LIN {X 0,Y 226.973,Z 1141.25,A -85,B 0,C 180,E1 10854.134,E2 10854.134} C_VEL
LIN {X 0,Y 235.059,Z 1134.942,A -85,B 0,C 180,E1 10847.384,E2 10847.384} C_VEL
LIN {X 0,Y 243.394,Z 1128.553,A -85,B 0,C 180,E1 10842.316,E2 10842.316} C_VEL
LIN {X 0,Y 253.409,Z 1120.828,A -85,B 0,C 180,E1 10837.527,E2 10837.527} C_VEL
LIN {X 0,Y 267.885,Z 1109.245,A -85,B 0,C 180,E1 10832.085,E2 10832.085} C_VEL
LIN {X 0,Y 280.211,Z 1098.882,A -85,B 0,C 180,E1 10828.333,E2 10828.333} C_VEL
LIN {X 0,Y 293.347,Z 1087.293,A -85,B 0,C 180,E1 10824.954,E2 10824.954} C_VEL
LIN {X 0,Y 310.134,Z 1071.349,A -85,B 0,C 180,E1 10821.295,E2 10821.295} C_VEL
LIN {X 0,Y 323.853,Z 1057.227,A -85,B 0,C 180,E1 10818.729,E2 10818.729} C_VEL
LIN {X 0,Y 337.044,Z 1042.652,A -85,B 0,C 180,E1 10816.547,E2 10816.547} C_VEL
LIN {X 0,Y 352.779,Z 1023.717,A -85,B 0,C 180,E1 10814.232,E2 10814.232} C_VEL
LIN {X 0,Y 366.214,Z 1005.755,A -85,B 0,C 180,E1 10812.456,E2 10812.456} C_VEL
LIN {X 0,Y 377.493,Z 989.298,A -85,B 0,C 180,E1 10811.087,E2 10811.087} C_VEL
LIN {X 0,Y 389.316,Z 970.374,A -85,B 0,C 180,E1 10809.759,E2 10809.759} C_VEL
LIN {X 0,Y 402.725,Z 946.04,A -85,B 0,C 180,E1 10808.363,E2 10808.363} C_VEL
LIN {X 0,Y 411.936,Z 927.031,A -85,B 0,C 180,E1 10807.468,E2 10807.468} C_VEL
LIN {X 0,Y 420.462,Z 907.175,A -85,B 0,C 180,E1 10806.669,E2 10806.669} C_VEL
LIN {X 0,Y 429.627,Z 882.607,A -85,B 0,C 180,E1 10805.851,E2 10805.851} C_VEL
LIN {X 0,Y 437.317,Z 856.996,A -85,B 0,C 180,E1 10805.178,E2 10805.178} C_VEL
LIN {X 0,Y 442.393,Z 836.475,A -85,B 0,C 180,E1 10804.748,E2 10804.748} C_VEL
LIN {X 0,Y 446.869,Z 813.721,A -85,B 0,C 180,E1 10804.357,E2 10804.357} C_VEL
LIN {X 0,Y 451.545,Z 778.74,A -85,B 0,C 180,E1 10803.872,E2 10803.872} C_VEL
LIN {X 0,Y 453.629,Z 760.255,A -85,B 0,C 180,E1 10803.626,E2 10803.626} C_VEL
LIN {X 0,Y 454.379,Z 752.732,A -85,B 0,C 180,E1 10803.403,E2 10803.403} C_VEL
LIN {X 0,Y 456.025,Z 733.241,A -85,B 0,C 180,E1 10802.357,E2 10802.357} C_VEL
LIN {X 0,Y 456.71,Z 726.771,A -85,B 0,C 180,E1 10802.178,E2 10802.178} C_VEL
LIN {X 0,Y 468.964,Z 621.482,A -85,B 0,C 180,E1 10800.794,E2 10800.794} C_VEL
LIN {X 0,Y 468.493,Z 619.747,A -85,B 0,C 180,E1 10797.798,E2 10797.798} C_VEL
LIN {X 0,Y 469.144,Z 622.007,A -85,B 0,C 180,E1 10794.232,E2 10794.232} C_VEL
LIN {X 0,Y 447.711,Z 806.552,A -85,B 0,C 180,E1 10791.736,E2 10791.736} C_VEL
LIN {X 0,Y 443.092,Z 833.793,A -85,B 0,C 180,E1 10791.332,E2 10791.332} C_VEL
LIN {X 0,Y 436.841,Z 859.788,A -85,B 0,C 180,E1 10790.9,E2 10790.9} C_VEL
LIN {X 0,Y 430.614,Z 880.919,A -85,B 0,C 180,E1 10790.485,E2 10790.485} C_VEL
LIN {X 0,Y 422.897,Z 903.181,A -85,B 0,C 180,E1 10789.937,E2 10789.937} C_VEL
LIN {X 0,Y 411.827,Z 930.087,A -85,B 0,C 180,E1 10789.097,E2 10789.097} C_VEL
LIN {X 0,Y 401.901,Z 950.938,A -85,B 0,C 180,E1 10788.281,E2 10788.281} C_VEL
LIN {X 0,Y 391.891,Z 969.818,A -85,B 0,C 180,E1 10787.395,E2 10787.395} C_VEL
LIN {X 0,Y 379.849,Z 990.376,A -85,B 0,C 180,E1 10786.24,E2 10786.24} C_VEL
LIN {X 0,Y 364.513,Z 1013.698,A -85,B 0,C 180,E1 10784.615,E2 10784.615} C_VEL
LIN {X 0,Y 351.656,Z 1031.443,A -85,B 0,C 180,E1 10783.091,E2 10783.091} C_VEL
LIN {X 0,Y 339.49,Z 1047.003,A -85,B 0,C 180,E1 10781.504,E2 10781.504} C_VEL
LIN {X 0,Y 325.202,Z 1064.029,A -85,B 0,C 180,E1 10779.424,E2 10779.424} C_VEL
LIN {X 0,Y 307.386,Z 1083.642,A -85,B 0,C 180,E1 10776.415,E2 10776.415} C_VEL
LIN {X 0,Y 293.416,Z 1097.967,A -85,B 0,C 180,E1 10773.665,E2 10773.665} C_VEL
LIN {X 0,Y 280.033,Z 1111.045,A -85,B 0,C 180,E1 10770.599,E2 10770.599} C_VEL
LIN {X 0,Y 265.034,Z 1125.203,A -85,B 0,C 180,E1 10766.485,E2 10766.485} C_VEL
LIN {X 0,Y 250.118,Z 1138.668,A -85,B 0,C 180,E1 10761.418,E2 10761.418} C_VEL
LIN {X 0,Y 239.086,Z 1148.595,A -85,B 0,C 180,E1 10756.691,E2 10756.691} C_VEL
LIN {X 0,Y 229.528,Z 1157.411,A -85,B 0,C 180,E1 10751.463,E2 10751.463} C_VEL
LIN {X 0,Y 219.97,Z 1166.782,A -85,B 0,C 180,E1 10744.308,E2 10744.308} C_VEL
LIN {X 0,Y 214.19,Z 1173.147,A -85,B 0,C 180,E1 10737.828,E2 10737.828} C_VEL
LIN {X 0,Y 210.917,Z 1177.583,A -85,B 0,C 180,E1 10731.994,E2 10731.994} C_VEL
LIN {X 0,Y 209.151,Z 1180.939,A -85,B 0,C 180,E1 10726.098,E2 10726.098} C_VEL
LIN {X 0,Y 208.563,Z 1183.075,A -85,B 0,C 180,E1 10720.638,E2 10720.638} C_VEL
LIN {X 0,Y 208.6,Z 1184.174,A -85,B 0,C 180,E1 10715.777,E2 10715.777} C_VEL
LIN {X 0,Y 208.736,Z 1184.477,A -85,B 0,C 180,E1 10711.098,E2 10711.098} C_VEL
LIN {X 0,Y 208.696,Z 1183.922,A -85,B 0,C 180,E1 10706.154,E2 10706.154} C_VEL
LIN {X 0,Y 208.612,Z 1182.339,A -85,B 0,C 180,E1 10700.886,E2 10700.886} C_VEL
LIN {X 0,Y 209.086,Z 1179.246,A -85,B 0,C 180,E1 10694.751,E2 10694.751} C_VEL
LIN {X 0,Y 210.519,Z 1175.309,A -85,B 0,C 180,E1 10689.132,E2 10689.132} C_VEL
LIN {X 0,Y 213.256,Z 1170.278,A -85,B 0,C 180,E1 10683.551,E2 10683.551} C_VEL
LIN {X 0,Y 217.415,Z 1164.128,A -85,B 0,C 180,E1 10678.071,E2 10678.071} C_VEL
LIN {X 0,Y 223.422,Z 1156.436,A -85,B 0,C 180,E1 10672.51,E2 10672.51} C_VEL
LIN {X 0,Y 233.164,Z 1145.065,A -85,B 0,C 180,E1 10665.998,E2 10665.998} C_VEL
LIN {X 0,Y 243.301,Z 1133.621,A -85,B 0,C 180,E1 10660.874,E2 10660.874} C_VEL
LIN {X 0,Y 253.371,Z 1122.401,A -85,B 0,C 180,E1 10656.767,E2 10656.767} C_VEL
LIN {X 0,Y 266.019,Z 1108.199,A -85,B 0,C 180,E1 10652.514,E2 10652.514} C_VEL
LIN {X 0,Y 280.155,Z 1091.564,A -85,B 0,C 180,E1 10648.572,E2 10648.572} C_VEL
LIN {X 0,Y 291.973,Z 1077.025,A -85,B 0,C 180,E1 10645.758,E2 10645.758} C_VEL
LIN {X 0,Y 303.945,Z 1061.531,A -85,B 0,C 180,E1 10643.251,E2 10643.251} C_VEL
LIN {X 0,Y 318.505,Z 1041.486,A -85,B 0,C 180,E1 10640.586,E2 10640.586} C_VEL
LIN {X 0,Y 331.631,Z 1021.599,A -85,B 0,C 180,E1 10638.456,E2 10638.456} C_VEL
LIN {X 0,Y 342.65,Z 1003.559,A -85,B 0,C 180,E1 10636.842,E2 10636.842} C_VEL
LIN {X 0,Y 354.044,Z 983.305,A -85,B 0,C 180,E1 10635.328,E2 10635.328} C_VEL
LIN {X 0,Y 366.538,Z 958.361,A -85,B 0,C 180,E1 10633.806,E2 10633.806} C_VEL
LIN {X 0,Y 375.614,Z 937.919,A -85,B 0,C 180,E1 10632.788,E2 10632.788} C_VEL
LIN {X 0,Y 383.742,Z 917.39,A -85,B 0,C 180,E1 10631.936,E2 10631.936} C_VEL
LIN {X 0,Y 392.509,Z 892.087,A -85,B 0,C 180,E1 10631.078,E2 10631.078} C_VEL
LIN {X 0,Y 399.826,Z 866.079,A -85,B 0,C 180,E1 10630.401,E2 10630.401} C_VEL
LIN {X 0,Y 404.934,Z 844.022,A -85,B 0,C 180,E1 10629.944,E2 10629.944} C_VEL
LIN {X 0,Y 409.416,Z 818.913,A -85,B 0,C 180,E1 10629.487,E2 10629.487} C_VEL
LIN {X 0,Y 413.661,Z 781.521,A -85,B 0,C 180,E1 10628.913,E2 10628.913} C_VEL
LIN {X 0,Y 432.506,Z 593.201,A -85,B 0,C 180,E1 10626.162,E2 10626.162} C_VEL
LIN {X 0,Y 429.414,Z 586.105,A -85,B 0,C 180,E1 10623.605,E2 10623.605} C_VEL
LIN {X 0,Y 427.117,Z 580.871,A -85,B 0,C 180,E1 10621.207,E2 10621.207} C_VEL
LIN {X 0,Y 425.896,Z 578.251,A -85,B 0,C 180,E1 10619.596,E2 10619.596} C_VEL
LIN {X 0,Y 424.641,Z 575.258,A -85,B 0,C 180,E1 10617.301,E2 10617.301} C_VEL
LIN {X 0,Y 423.647,Z 573.176,A -85,B 0,C 180,E1 10613.223,E2 10613.223} C_VEL
LIN {X 0,Y 423.893,Z 573.926,A -85,B 0,C 180,E1 10610.496,E2 10610.496} C_VEL
LIN {X 0,Y 424.964,Z 575.871,A -85,B 0,C 180,E1 10607.705,E2 10607.705} C_VEL
LIN {X 0,Y 426.778,Z 579.948,A -85,B 0,C 180,E1 10604.926,E2 10604.926} C_VEL
LIN {X 0,Y 429.137,Z 585.108,A -85,B 0,C 180,E1 10602.368,E2 10602.368} C_VEL
LIN {X 0,Y 430.931,Z 589.439,A -85,B 0,C 180,E1 10600.767,E2 10600.767} C_VEL
LIN {X 0,Y 409.317,Z 799.134,A -85,B 0,C 180,E1 10597.801,E2 10597.801} C_VEL
LIN {X 0,Y 405.219,Z 825.67,A -85,B 0,C 180,E1 10597.343,E2 10597.343} C_VEL
LIN {X 0,Y 399.741,Z 850.636,A -85,B 0,C 180,E1 10596.777,E2 10596.777} C_VEL
LIN {X 0,Y 394.029,Z 871.901,A -85,B 0,C 180,E1 10596.174,E2 10596.174} C_VEL
LIN {X 0,Y 386.657,Z 895.114,A -85,B 0,C 180,E1 10595.36,E2 10595.36} C_VEL
LIN {X 0,Y 377.297,Z 919.717,A -85,B 0,C 180,E1 10594.292,E2 10594.292} C_VEL
LIN {X 0,Y 368.832,Z 939.096,A -85,B 0,C 180,E1 10593.282,E2 10593.282} C_VEL
LIN {X 0,Y 359.283,Z 958.656,A -85,B 0,C 180,E1 10592.077,E2 10592.077} C_VEL
LIN {X 0,Y 346.794,Z 981.508,A -85,B 0,C 180,E1 10590.373,E2 10590.373} C_VEL
LIN {X 0,Y 334.96,Z 1000.727,A -85,B 0,C 180,E1 10588.617,E2 10588.617} C_VEL
LIN {X 0,Y 323.806,Z 1017.378,A -85,B 0,C 180,E1 10586.804,E2 10586.804} C_VEL
LIN {X 0,Y 310.836,Z 1035.283,A -85,B 0,C 180,E1 10584.47,E2 10584.47} C_VEL
LIN {X 0,Y 296.991,Z 1052.66,A -85,B 0,C 180,E1 10581.667,E2 10581.667} C_VEL
LIN {X 0,Y 285.132,Z 1066.573,A -85,B 0,C 180,E1 10578.932,E2 10578.932} C_VEL
LIN {X 0,Y 273.308,Z 1079.709,A -85,B 0,C 180,E1 10575.81,E2 10575.81} C_VEL
LIN {X 0,Y 258.957,Z 1094.789,A -85,B 0,C 180,E1 10571.319,E2 10571.319} C_VEL
LIN {X 0,Y 248.09,Z 1105.699,A -85,B 0,C 180,E1 10567.195,E2 10567.195} C_VEL
LIN {X 0,Y 238.437,Z 1115.241,A -85,B 0,C 180,E1 10562.748,E2 10562.748} C_VEL
LIN {X 0,Y 228.33,Z 1125.281,A -85,B 0,C 180,E1 10556.81,E2 10556.81} C_VEL
LIN {X 0,Y 220.905,Z 1132.814,A -85,B 0,C 180,E1 10550.951,E2 10550.951} C_VEL
LIN {X 0,Y 215.987,Z 1138.253,A -85,B 0,C 180,E1 10545.575,E2 10545.575} C_VEL
LIN {X 0,Y 212.122,Z 1143.214,A -85,B 0,C 180,E1 10539.222,E2 10539.222} C_VEL
LIN {X 0,Y 209.809,Z 1146.998,A -85,B 0,C 180,E1 10532.185,E2 10532.185} C_VEL
LIN {X 0,Y 209.054,Z 1148.977,A -85,B 0,C 180,E1 10526.435,E2 10526.435} C_VEL
LIN {X 0,Y 208.923,Z 1149.951,A -85,B 0,C 180,E1 10521.468,E2 10521.468} C_VEL
LIN {X 0,Y 209.12,Z 1150.229,A -85,B 0,C 180,E1 10516.08,E2 10516.08} C_VEL
LIN {X 0,Y 209.869,Z 1149.696,A -85,B 0,C 180,E1 10510.622,E2 10510.622} C_VEL
LIN {X 0,Y 211.518,Z 1148.307,A -85,B 0,C 180,E1 10505.121,E2 10505.121} C_VEL
LIN {X 0,Y 214.52,Z 1145.926,A -85,B 0,C 180,E1 10499.467,E2 10499.467} C_VEL
LIN {X 0,Y 219.826,Z 1141.985,A -85,B 0,C 180,E1 10493.102,E2 10493.102} C_VEL
LIN {X 0,Y 228.359,Z 1135.76,A -85,B 0,C 180,E1 10486.227,E2 10486.227} C_VEL
LIN {X 0,Y 237.216,Z 1129.338,A -85,B 0,C 180,E1 10481.02,E2 10481.02} C_VEL
LIN {X 0,Y 247.177,Z 1122.02,A -85,B 0,C 180,E1 10476.392,E2 10476.392} C_VEL
LIN {X 0,Y 260.95,Z 1111.6,A -85,B 0,C 180,E1 10471.301,E2 10471.301} C_VEL
LIN {X 0,Y 275.102,Z 1100.135,A -85,B 0,C 180,E1 10467.07,E2 10467.07} C_VEL
LIN {X 0,Y 287.664,Z 1089.441,A -85,B 0,C 180,E1 10463.917,E2 10463.917} C_VEL
LIN {X 0,Y 303.29,Z 1075.322,A -85,B 0,C 180,E1 10460.567,E2 10460.567} C_VEL
LIN {X 0,Y 319.008,Z 1059.686,A -85,B 0,C 180,E1 10457.67,E2 10457.67} C_VEL
LIN {X 0,Y 332.216,Z 1045.543,A -85,B 0,C 180,E1 10455.538,E2 10455.538} C_VEL
LIN {X 0,Y 345.206,Z 1030.544,A -85,B 0,C 180,E1 10453.652,E2 10453.652} C_VEL
LIN {X 0,Y 360.841,Z 1010.795,A -85,B 0,C 180,E1 10451.617,E2 10451.617} C_VEL
LIN {X 0,Y 374.22,Z 991.831,A -85,B 0,C 180,E1 10450.033,E2 10450.033} C_VEL
LIN {X 0,Y 385.523,Z 974.223,A -85,B 0,C 180,E1 10448.802,E2 10448.802} C_VEL
LIN {X 0,Y 396.927,Z 954.579,A -85,B 0,C 180,E1 10447.65,E2 10447.65} C_VEL
LIN {X 0,Y 409.069,Z 930.705,A -85,B 0,C 180,E1 10446.497,E2 10446.497} C_VEL
LIN {X 0,Y 417.999,Z 910.507,A -85,B 0,C 180,E1 10445.687,E2 10445.687} C_VEL
LIN {X 0,Y 425.879,Z 890.172,A -85,B 0,C 180,E1 10445.006,E2 10445.006} C_VEL
LIN {X 0,Y 433.214,Z 868.163,A -85,B 0,C 180,E1 10444.397,E2 10444.397} C_VEL
LIN {X 0,Y 440.387,Z 841.427,A -85,B 0,C 180,E1 10443.801,E2 10443.801} C_VEL
LIN {X 0,Y 445.099,Z 818.79,A -85,B 0,C 180,E1 10443.407,E2 10443.407} C_VEL
LIN {X 0,Y 448.671,Z 795.814,A -85,B 0,C 180,E1 10443.083,E2 10443.083} C_VEL
LIN {X 0,Y 456.71,Z 726.771,A -85,B 0,C 180,E1 10442.178,E2 10442.178} C_VEL
LIN {X 0,Y 457.501,Z 719.251,A -85,B 0,C 180,E1 10441.956,E2 10441.956} C_VEL
LIN {X 0,Y 459.355,Z 699.763,A -85,B 0,C 180,E1 10440.922,E2 10440.922} C_VEL
LIN {X 0,Y 460.075,Z 693.295,A -85,B 0,C 180,E1 10440.746,E2 10440.746} C_VEL
LIN {X 0,Y 467.717,Z 628.788,A -85,B 0,C 180,E1 10439.908,E2 10439.908} C_VEL
LIN {X 0,Y 467.51,Z 627.71,A -85,B 0,C 180,E1 10437.671,E2 10437.671} C_VEL
LIN {X 0,Y 467.821,Z 629.471,A -85,B 0,C 180,E1 10435.114,E2 10435.114} C_VEL
LIN {X 0,Y 446.95,Z 806.235,A -85,B 0,C 180,E1 10432.764,E2 10432.764} C_VEL
LIN {X 0,Y 442.26,Z 833.504,A -85,B 0,C 180,E1 10432.37,E2 10432.37} C_VEL
LIN {X 0,Y 436.004,Z 859.276,A -85,B 0,C 180,E1 10431.956,E2 10431.956} C_VEL
LIN {X 0,Y 429.602,Z 880.773,A -85,B 0,C 180,E1 10431.551,E2 10431.551} C_VEL
LIN {X 0,Y 421.288,Z 904.409,A -85,B 0,C 180,E1 10430.988,E2 10430.988} C_VEL
LIN {X 0,Y 410.38,Z 930.338,A -85,B 0,C 180,E1 10430.201,E2 10430.201} C_VEL
LIN {X 0,Y 400.723,Z 950.357,A -85,B 0,C 180,E1 10429.446,E2 10429.446} C_VEL
LIN {X 0,Y 390.199,Z 969.916,A -85,B 0,C 180,E1 10428.559,E2 10428.559} C_VEL
LIN {X 0,Y 376.647,Z 992.59,A -85,B 0,C 180,E1 10427.311,E2 10427.311} C_VEL
LIN {X 0,Y 361.978,Z 1014.221,A -85,B 0,C 180,E1 10425.821,E2 10425.821} C_VEL
LIN {X 0,Y 349.423,Z 1031.208,A -85,B 0,C 180,E1 10424.396,E2 10424.396} C_VEL
LIN {X 0,Y 336.676,Z 1047.159,A -85,B 0,C 180,E1 10422.809,E2 10422.809} C_VEL
LIN {X 0,Y 320.16,Z 1066.361,A -85,B 0,C 180,E1 10420.478,E2 10420.478} C_VEL
LIN {X 0,Y 303.29,Z 1084.191,A -85,B 0,C 180,E1 10417.72,E2 10417.72} C_VEL
LIN {X 0,Y 289.027,Z 1098.357,A -85,B 0,C 180,E1 10415.007,E2 10415.007} C_VEL
LIN {X 0,Y 274.574,Z 1111.996,A -85,B 0,C 180,E1 10411.793,E2 10411.793} C_VEL
LIN {X 0,Y 256.613,Z 1128.095,A -85,B 0,C 180,E1 10406.9,E2 10406.9} C_VEL
LIN {X 0,Y 244.029,Z 1138.962,A -85,B 0,C 180,E1 10402.644,E2 10402.644} C_VEL
LIN {X 0,Y 232.682,Z 1148.677,A -85,B 0,C 180,E1 10397.904,E2 10397.904} C_VEL
LIN {X 0,Y 221.195,Z 1158.795,A -85,B 0,C 180,E1 10391.643,E2 10391.643} C_VEL
LIN {X 0,Y 212.147,Z 1167.063,A -85,B 0,C 180,E1 10384.77,E2 10384.77} C_VEL
LIN {X 0,Y 206.612,Z 1172.797,A -85,B 0,C 180,E1 10378.626,E2 10378.626} C_VEL
LIN {X 0,Y 203.12,Z 1177.165,A -85,B 0,C 180,E1 10372.579,E2 10372.579} C_VEL
LIN {X 0,Y 201.217,Z 1180.457,A -85,B 0,C 180,E1 10366.451,E2 10366.451} C_VEL
LIN {X 0,Y 200.579,Z 1182.569,A -85,B 0,C 180,E1 10360.629,E2 10360.629} C_VEL
LIN {X 0,Y 200.625,Z 1183.558,A -85,B 0,C 180,E1 10355.721,E2 10355.721} C_VEL
LIN {X 0,Y 200.763,Z 1183.806,A -85,B 0,C 180,E1 10351.142,E2 10351.142} C_VEL
LIN {X 0,Y 200.725,Z 1183.298,A -85,B 0,C 180,E1 10346.287,E2 10346.287} C_VEL
LIN {X 0,Y 200.635,Z 1181.675,A -85,B 0,C 180,E1 10340.667,E2 10340.667} C_VEL
LIN {X 0,Y 201.143,Z 1178.661,A -85,B 0,C 180,E1 10334.43,E2 10334.43} C_VEL
LIN {X 0,Y 202.799,Z 1174.51,A -85,B 0,C 180,E1 10328.299,E2 10328.299} C_VEL
LIN {X 0,Y 205.793,Z 1169.444,A -85,B 0,C 180,E1 10322.512,E2 10322.512} C_VEL
LIN {X 0,Y 210.383,Z 1163.151,A -85,B 0,C 180,E1 10316.771,E2 10316.771} C_VEL
LIN {X 0,Y 217.499,Z 1154.673,A -85,B 0,C 180,E1 10310.564,E2 10310.564} C_VEL
LIN {X 0,Y 227.982,Z 1143.073,A -85,B 0,C 180,E1 10304.007,E2 10304.007} C_VEL
LIN {X 0,Y 237.776,Z 1132.582,A -85,B 0,C 180,E1 10299.311,E2 10299.311} C_VEL
LIN {X 0,Y 248.459,Z 1121.18,A -85,B 0,C 180,E1 10295.134,E2 10295.134} C_VEL
LIN {X 0,Y 262.566,Z 1105.876,A -85,B 0,C 180,E1 10290.615,E2 10290.615} C_VEL
LIN {X 0,Y 276.089,Z 1090.381,A -85,B 0,C 180,E1 10287.015,E2 10287.015} C_VEL
LIN {X 0,Y 288.342,Z 1075.724,A -85,B 0,C 180,E1 10284.22,E2 10284.22} C_VEL
LIN {X 0,Y 301.209,Z 1059.48,A -85,B 0,C 180,E1 10281.651,E2 10281.651} C_VEL
LIN {X 0,Y 317.04,Z 1037.853,A -85,B 0,C 180,E1 10278.895,E2 10278.895} C_VEL
LIN {X 0,Y 328.517,Z 1020.788,A -85,B 0,C 180,E1 10277.124,E2 10277.124} C_VEL
LIN {X 0,Y 339.431,Z 1003.265,A -85,B 0,C 180,E1 10275.584,E2 10275.584} C_VEL
LIN {X 0,Y 350.593,Z 983.815,A -85,B 0,C 180,E1 10274.153,E2 10274.153} C_VEL
LIN {X 0,Y 363.728,Z 958.14,A -85,B 0,C 180,E1 10272.614,E2 10272.614} C_VEL
LIN {X 0,Y 373.21,Z 937.079,A -85,B 0,C 180,E1 10271.592,E2 10271.592} C_VEL
LIN {X 0,Y 381.186,Z 917.222,A -85,B 0,C 180,E1 10270.791,E2 10270.791} C_VEL
LIN {X 0,Y 390.069,Z 891.978,A -85,B 0,C 180,E1 10269.956,E2 10269.956} C_VEL
LIN {X 0,Y 397.537,Z 865.841,A -85,B 0,C 180,E1 10269.294,E2 10269.294} C_VEL
LIN {X 0,Y 402.702,Z 843.836,A -85,B 0,C 180,E1 10268.849,E2 10268.849} C_VEL
LIN {X 0,Y 407.164,Z 819.265,A -85,B 0,C 180,E1 10268.411,E2 10268.411} C_VEL
LIN {X 0,Y 411.44,Z 782.791,A -85,B 0,C 180,E1 10267.856,E2 10267.856} C_VEL
LIN {X 0,Y 430.21,Z 598.71,A -85,B 0,C 180,E1 10265.201,E2 10265.201} C_VEL
LIN {X 0,Y 426.925,Z 590.926,A -85,B 0,C 180,E1 10262.148,E2 10262.148} C_VEL
LIN {X 0,Y 424.946,Z 586.384,A -85,B 0,C 180,E1 10259.666,E2 10259.666} C_VEL
LIN {X 0,Y 423.588,Z 583.13,A -85,B 0,C 180,E1 10257.159,E2 10257.159} C_VEL
LIN {X 0,Y 422.666,Z 581.091,A -85,B 0,C 180,E1 10253.07,E2 10253.07} C_VEL
LIN {X 0,Y 423.018,Z 582.127,A -85,B 0,C 180,E1 10250.064,E2 10250.064} C_VEL
LIN {X 0,Y 423.915,Z 583.794,A -85,B 0,C 180,E1 10247.813,E2 10247.813} C_VEL
LIN {X 0,Y 425.638,Z 587.792,A -85,B 0,C 180,E1 10245.094,E2 10245.094} C_VEL
LIN {X 0,Y 427.801,Z 592.687,A -85,B 0,C 180,E1 10242.662,E2 10242.662} C_VEL
LIN {X 0,Y 428.75,Z 595.232,A -85,B 0,C 180,E1 10241.736,E2 10241.736} C_VEL
LIN {X 0,Y 407.291,Z 799.62,A -85,B 0,C 180,E1 10238.885,E2 10238.885} C_VEL
LIN {X 0,Y 403.105,Z 826.259,A -85,B 0,C 180,E1 10238.433,E2 10238.433} C_VEL
LIN {X 0,Y 397.576,Z 851.112,A -85,B 0,C 180,E1 10237.883,E2 10237.883} C_VEL
LIN {X 0,Y 391.809,Z 872.298,A -85,B 0,C 180,E1 10237.296,E2 10237.296} C_VEL
LIN {X 0,Y 384.741,Z 894.289,A -85,B 0,C 180,E1 10236.544,E2 10236.544} C_VEL
LIN {X 0,Y 374.818,Z 920.138,A -85,B 0,C 180,E1 10235.456,E2 10235.456} C_VEL
LIN {X 0,Y 366.214,Z 939.527,A -85,B 0,C 180,E1 10234.468,E2 10234.468} C_VEL
LIN {X 0,Y 356.904,Z 958.318,A -85,B 0,C 180,E1 10233.338,E2 10233.338} C_VEL
LIN {X 0,Y 344.579,Z 980.681,A -85,B 0,C 180,E1 10231.722,E2 10231.722} C_VEL
LIN {X 0,Y 331.718,Z 1001.191,A -85,B 0,C 180,E1 10229.89,E2 10229.89} C_VEL
LIN {X 0,Y 320.326,Z 1017.853,A -85,B 0,C 180,E1 10228.104,E2 10228.104} C_VEL
LIN {X 0,Y 307.053,Z 1035.77,A -85,B 0,C 180,E1 10225.802,E2 10225.802} C_VEL
LIN {X 0,Y 292.855,Z 1053.163,A -85,B 0,C 180,E1 10223.027,E2 10223.027} C_VEL
LIN {X 0,Y 280.662,Z 1067.092,A -85,B 0,C 180,E1 10220.309,E2 10220.309} C_VEL
LIN {X 0,Y 268.468,Z 1080.248,A -85,B 0,C 180,E1 10217.196,E2 10217.196} C_VEL
LIN {X 0,Y 253.611,Z 1095.343,A -85,B 0,C 180,E1 10212.696,E2 10212.696} C_VEL
LIN {X 0,Y 242.311,Z 1106.262,A -85,B 0,C 180,E1 10208.541,E2 10208.541} C_VEL
LIN {X 0,Y 232.232,Z 1115.814,A -85,B 0,C 180,E1 10204.035,E2 10204.035} C_VEL
LIN {X 0,Y 221.615,Z 1125.875,A -85,B 0,C 180,E1 10197.983,E2 10197.983} C_VEL
LIN {X 0,Y 213.769,Z 1133.416,A -85,B 0,C 180,E1 10191.974,E2 10191.974} C_VEL
LIN {X 0,Y 208.327,Z 1139.099,A -85,B 0,C 180,E1 10186.163,E2 10186.163} C_VEL
LIN {X 0,Y 204.017,Z 1144.394,A -85,B 0,C 180,E1 10179.023,E2 10179.023} C_VEL
LIN {X 0,Y 201.788,Z 1147.844,A -85,B 0,C 180,E1 10171.988,E2 10171.988} C_VEL
LIN {X 0,Y 201.09,Z 1149.618,A -85,B 0,C 180,E1 10166.579,E2 10166.579} C_VEL
LIN {X 0,Y 200.948,Z 1150.603,A -85,B 0,C 180,E1 10161.415,E2 10161.415} C_VEL
LIN {X 0,Y 201.16,Z 1150.9,A -85,B 0,C 180,E1 10155.903,E2 10155.903} C_VEL
LIN {X 0,Y 201.991,Z 1150.381,A -85,B 0,C 180,E1 10150.142,E2 10150.142} C_VEL
LIN {X 0,Y 203.802,Z 1149.008,A -85,B 0,C 180,E1 10144.422,E2 10144.422} C_VEL
LIN {X 0,Y 207.053,Z 1146.645,A -85,B 0,C 180,E1 10138.565,E2 10138.565} C_VEL
LIN {X 0,Y 212.514,Z 1142.873,A -85,B 0,C 180,E1 10132.228,E2 10132.228} C_VEL
LIN {X 0,Y 221.829,Z 1136.527,A -85,B 0,C 180,E1 10124.956,E2 10124.956} C_VEL
LIN {X 0,Y 231.165,Z 1130.124,A -85,B 0,C 180,E1 10119.655,E2 10119.655} C_VEL
LIN {X 0,Y 241.605,Z 1122.828,A -85,B 0,C 180,E1 10114.975,E2 10114.975} C_VEL
LIN {X 0,Y 255.949,Z 1112.45,A -85,B 0,C 180,E1 10109.86,E2 10109.86} C_VEL
LIN {X 0,Y 270.732,Z 1100.903,A -85,B 0,C 180,E1 10105.602,E2 10105.602} C_VEL
LIN {X 0,Y 284.397,Z 1089.629,A -85,B 0,C 180,E1 10102.316,E2 10102.316} C_VEL
LIN {X 0,Y 300.418,Z 1075.524,A -85,B 0,C 180,E1 10099.037,E2 10099.037} C_VEL
LIN {X 0,Y 316.53,Z 1059.841,A -85,B 0,C 180,E1 10096.203,E2 10096.203} C_VEL
LIN {X 0,Y 330.37,Z 1045.312,A -85,B 0,C 180,E1 10094.073,E2 10094.073} C_VEL
LIN {X 0,Y 344.627,Z 1029.094,A -85,B 0,C 180,E1 10092.114,E2 10092.114} C_VEL
LIN {X 0,Y 360.588,Z 1008.926,A -85,B 0,C 180,E1 10090.145,E2 10090.145} C_VEL
LIN {X 0,Y 372.562,Z 992.172,A -85,B 0,C 180,E1 10088.8,E2 10088.8} C_VEL
LIN {X 0,Y 384.302,Z 974.122,A -85,B 0,C 180,E1 10087.578,E2 10087.578} C_VEL
LIN {X 0,Y 397.361,Z 951.794,A -85,B 0,C 180,E1 10086.323,E2 10086.323} C_VEL
LIN {X 0,Y 408.69,Z 929.299,A -85,B 0,C 180,E1 10085.3,E2 10085.3} C_VEL
LIN {X 0,Y 417.262,Z 910.037,A -85,B 0,C 180,E1 10084.561,E2 10084.561} C_VEL
LIN {X 0,Y 425.417,Z 889.098,A -85,B 0,C 180,E1 10083.885,E2 10083.885} C_VEL
LIN {X 0,Y 433.932,Z 863.135,A -85,B 0,C 180,E1 10083.21,E2 10083.21} C_VEL
LIN {X 0,Y 440.01,Z 839.798,A -85,B 0,C 180,E1 10082.728,E2 10082.728} C_VEL
LIN {X 0,Y 444.534,Z 817.979,A -85,B 0,C 180,E1 10082.364,E2 10082.364} C_VEL
LIN {X 0,Y 448.418,Z 792.688,A -85,B 0,C 180,E1 10082.018,E2 10082.018} C_VEL
LIN {X 0,Y 460.075,Z 693.295,A -85,B 0,C 180,E1 10080.746,E2 10080.746} C_VEL
LIN {X 0,Y 460.91,Z 685.778,A -85,B 0,C 180,E1 10080.527,E2 10080.527} C_VEL
LIN {X 0,Y 462.968,Z 666.296,A -85,B 0,C 180,E1 10079.507,E2 10079.507} C_VEL
LIN {X 0,Y 463.72,Z 659.833,A -85,B 0,C 180,E1 10079.331,E2 10079.331} C_VEL
LIN {X 0,Y 466.579,Z 636.14,A -85,B 0,C 180,E1 10079.018,E2 10079.018} C_VEL
LIN {X 0,Y 466.529,Z 635.734,A -85,B 0,C 180,E1 10077.42,E2 10077.42} C_VEL
LIN {X 0,Y 466.63,Z 636.753,A -85,B 0,C 180,E1 10076.005,E2 10076.005} C_VEL
LIN {X 0,Y 446.333,Z 805.917,A -85,B 0,C 180,E1 10073.796,E2 10073.796} C_VEL
LIN {X 0,Y 441.573,Z 833.214,A -85,B 0,C 180,E1 10073.412,E2 10073.412} C_VEL
LIN {X 0,Y 435.265,Z 858.944,A -85,B 0,C 180,E1 10073.013,E2 10073.013} C_VEL
LIN {X 0,Y 428.763,Z 880.555,A -85,B 0,C 180,E1 10072.623,E2 10072.623} C_VEL
LIN {X 0,Y 420.441,Z 903.961,A -85,B 0,C 180,E1 10072.089,E2 10072.089} C_VEL
LIN {X 0,Y 409.604,Z 929.488,A -85,B 0,C 180,E1 10071.348,E2 10071.348} C_VEL
LIN {X 0,Y 399.833,Z 949.542,A -85,B 0,C 180,E1 10070.626,E2 10070.626} C_VEL
LIN {X 0,Y 389.416,Z 968.708,A -85,B 0,C 180,E1 10069.795,E2 10069.795} C_VEL
LIN {X 0,Y 376.755,Z 989.7,A -85,B 0,C 180,E1 10068.697,E2 10068.697} C_VEL
LIN {X 0,Y 360.95,Z 1012.913,A -85,B 0,C 180,E1 10067.179,E2 10067.179} C_VEL
LIN {X 0,Y 348.09,Z 1030.057,A -85,B 0,C 180,E1 10065.799,E2 10065.799} C_VEL
LIN {X 0,Y 334.589,Z 1046.658,A -85,B 0,C 180,E1 10064.204,E2 10064.204} C_VEL
LIN {X 0,Y 317.634,Z 1065.958,A -85,B 0,C 180,E1 10061.924,E2 10061.924} C_VEL
LIN {X 0,Y 300.456,Z 1083.661,A -85,B 0,C 180,E1 10059.247,E2 10059.247} C_VEL
LIN {X 0,Y 286.333,Z 1097.314,A -85,B 0,C 180,E1 10056.691,E2 10056.691} C_VEL
LIN {X 0,Y 271.289,Z 1111.076,A -85,B 0,C 180,E1 10053.514,E2 10053.514} C_VEL
LIN {X 0,Y 253.208,Z 1126.741,A -85,B 0,C 180,E1 10048.848,E2 10048.848} C_VEL
LIN {X 0,Y 239.564,Z 1138.023,A -85,B 0,C 180,E1 10044.475,E2 10044.475} C_VEL
LIN {X 0,Y 227.772,Z 1147.626,A -85,B 0,C 180,E1 10039.802,E2 10039.802} C_VEL
LIN {X 0,Y 215.945,Z 1157.391,A -85,B 0,C 180,E1 10033.753,E2 10033.753} C_VEL
LIN {X 0,Y 205.593,Z 1166.221,A -85,B 0,C 180,E1 10026.393,E2 10026.393} C_VEL
LIN {X 0,Y 199.533,Z 1171.982,A -85,B 0,C 180,E1 10020.073,E2 10020.073} C_VEL
LIN {X 0,Y 195.626,Z 1176.385,A -85,B 0,C 180,E1 10013.806,E2 10013.806} C_VEL
LIN {X 0,Y 193.421,Z 1179.701,A -85,B 0,C 180,E1 10007.447,E2 10007.447} C_VEL
LIN {X 0,Y 192.617,Z 1181.848,A -85,B 0,C 180,E1 10001.377,E2 10001.377} C_VEL
LIN {X 0,Y 192.632,Z 1182.871,A -85,B 0,C 180,E1 9996.258,E2 9996.258} C_VEL
LIN {X 0,Y 192.784,Z 1183.152,A -85,B 0,C 180,E1 9991.486,E2 9991.486} C_VEL
LIN {X 0,Y 192.755,Z 1182.673,A -85,B 0,C 180,E1 9986.431,E2 9986.431} C_VEL
LIN {X 0,Y 192.654,Z 1181.139,A -85,B 0,C 180,E1 9980.742,E2 9980.742} C_VEL
LIN {X 0,Y 193.205,Z 1178.076,A -85,B 0,C 180,E1 9974.081,E2 9974.081} C_VEL
LIN {X 0,Y 194.994,Z 1173.941,A -85,B 0,C 180,E1 9967.701,E2 9967.701} C_VEL
LIN {X 0,Y 198.195,Z 1168.886,A -85,B 0,C 180,E1 9961.692,E2 9961.692} C_VEL
LIN {X 0,Y 203,Z 1162.712,A -85,B 0,C 180,E1 9955.841,E2 9955.841} C_VEL
LIN {X 0,Y 209.81,Z 1154.996,A -85,B 0,C 180,E1 9949.958,E2 9949.958} C_VEL
LIN {X 0,Y 220.703,Z 1143.575,A -85,B 0,C 180,E1 9943.165,E2 9943.165} C_VEL
LIN {X 0,Y 231.343,Z 1132.661,A -85,B 0,C 180,E1 9938.132,E2 9938.132} C_VEL
LIN {X 0,Y 242.264,Z 1121.478,A -85,B 0,C 180,E1 9933.947,E2 9933.947} C_VEL
LIN {X 0,Y 255.61,Z 1107.55,A -85,B 0,C 180,E1 9929.729,E2 9929.729} C_VEL
LIN {X 0,Y 270.847,Z 1090.791,A -85,B 0,C 180,E1 9925.744,E2 9925.744} C_VEL
LIN {X 0,Y 283.408,Z 1076.234,A -85,B 0,C 180,E1 9922.957,E2 9922.957} C_VEL
LIN {X 0,Y 295.777,Z 1061.073,A -85,B 0,C 180,E1 9920.548,E2 9920.548} C_VEL
LIN {X 0,Y 310.261,Z 1042.152,A -85,B 0,C 180,E1 9918.071,E2 9918.071} C_VEL
LIN {X 0,Y 324.837,Z 1021.116,A -85,B 0,C 180,E1 9915.871,E2 9915.871} C_VEL
LIN {X 0,Y 336.38,Z 1002.969,A -85,B 0,C 180,E1 9914.304,E2 9914.304} C_VEL
LIN {X 0,Y 347.732,Z 983.527,A -85,B 0,C 180,E1 9912.904,E2 9912.904} C_VEL
LIN {X 0,Y 361.077,Z 957.9,A -85,B 0,C 180,E1 9911.404,E2 9911.404} C_VEL
LIN {X 0,Y 370.657,Z 936.97,A -85,B 0,C 180,E1 9910.413,E2 9910.413} C_VEL
LIN {X 0,Y 378.785,Z 917.055,A -85,B 0,C 180,E1 9909.631,E2 9909.631} C_VEL
LIN {X 0,Y 387.548,Z 892.529,A -85,B 0,C 180,E1 9908.84,E2 9908.84} C_VEL
LIN {X 0,Y 395.252,Z 866.169,A -85,B 0,C 180,E1 9908.187,E2 9908.187} C_VEL
LIN {X 0,Y 400.55,Z 843.978,A -85,B 0,C 180,E1 9907.749,E2 9907.749} C_VEL
LIN {X 0,Y 404.913,Z 820.475,A -85,B 0,C 180,E1 9907.337,E2 9907.337} C_VEL
LIN {X 0,Y 409.287,Z 784.776,A -85,B 0,C 180,E1 9906.798,E2 9906.798} C_VEL
LIN {X 0,Y 428.003,Z 604.35,A -85,B 0,C 180,E1 9904.22,E2 9904.22} C_VEL
LIN {X 0,Y 425.263,Z 597.533,A -85,B 0,C 180,E1 9901.415,E2 9901.415} C_VEL
LIN {X 0,Y 423.716,Z 593.982,A -85,B 0,C 180,E1 9899.324,E2 9899.324} C_VEL
LIN {X 0,Y 422.524,Z 590.981,A -85,B 0,C 180,E1 9896.984,E2 9896.984} C_VEL
LIN {X 0,Y 421.688,Z 589.03,A -85,B 0,C 180,E1 9893.054,E2 9893.054} C_VEL
LIN {X 0,Y 422.043,Z 590.1,A -85,B 0,C 180,E1 9890.041,E2 9890.041} C_VEL
LIN {X 0,Y 422.838,Z 591.615,A -85,B 0,C 180,E1 9887.989,E2 9887.989} C_VEL
LIN {X 0,Y 424.45,Z 595.507,A -85,B 0,C 180,E1 9885.331,E2 9885.331} C_VEL
LIN {X 0,Y 426.477,Z 600.266,A -85,B 0,C 180,E1 9882.958,E2 9882.958} C_VEL
LIN {X 0,Y 426.691,Z 601.038,A -85,B 0,C 180,E1 9882.715,E2 9882.715} C_VEL
LIN {X 0,Y 405.423,Z 799.995,A -85,B 0,C 180,E1 9879.981,E2 9879.981} C_VEL
LIN {X 0,Y 401.164,Z 826.685,A -85,B 0,C 180,E1 9879.538,E2 9879.538} C_VEL
LIN {X 0,Y 395.568,Z 851.502,A -85,B 0,C 180,E1 9879.002,E2 9879.002} C_VEL
LIN {X 0,Y 389.738,Z 872.631,A -85,B 0,C 180,E1 9878.431,E2 9878.431} C_VEL
LIN {X 0,Y 382.568,Z 894.653,A -85,B 0,C 180,E1 9877.697,E2 9877.697} C_VEL
LIN {X 0,Y 372.496,Z 920.545,A -85,B 0,C 180,E1 9876.635,E2 9876.635} C_VEL
LIN {X 0,Y 363.756,Z 939.958,A -85,B 0,C 180,E1 9875.671,E2 9875.671} C_VEL
LIN {X 0,Y 354.294,Z 958.756,A -85,B 0,C 180,E1 9874.565,E2 9874.565} C_VEL
LIN {X 0,Y 341.75,Z 981.135,A -85,B 0,C 180,E1 9872.983,E2 9872.983} C_VEL
LIN {X 0,Y 328.644,Z 1001.656,A -85,B 0,C 180,E1 9871.187,E2 9871.187} C_VEL
LIN {X 0,Y 317.397,Z 1017.798,A -85,B 0,C 180,E1 9869.494,E2 9869.494} C_VEL
LIN {X 0,Y 304.921,Z 1034.323,A -85,B 0,C 180,E1 9867.428,E2 9867.428} C_VEL
LIN {X 0,Y 288.888,Z 1053.666,A -85,B 0,C 180,E1 9864.424,E2 9864.424} C_VEL
LIN {X 0,Y 276.358,Z 1067.606,A -85,B 0,C 180,E1 9861.73,E2 9861.73} C_VEL
LIN {X 0,Y 264.432,Z 1080.107,A -85,B 0,C 180,E1 9858.803,E2 9858.803} C_VEL
LIN {X 0,Y 250.197,Z 1094.268,A -85,B 0,C 180,E1 9854.696,E2 9854.696} C_VEL
LIN {X 0,Y 237.205,Z 1106.343,A -85,B 0,C 180,E1 9850.159,E2 9850.159} C_VEL
LIN {X 0,Y 227.095,Z 1115.525,A -85,B 0,C 180,E1 9845.843,E2 9845.843} C_VEL
LIN {X 0,Y 216.967,Z 1124.671,A -85,B 0,C 180,E1 9840.458,E2 9840.458} C_VEL
LIN {X 0,Y 207.319,Z 1133.451,A -85,B 0,C 180,E1 9833.596,E2 9833.596} C_VEL
LIN {X 0,Y 201.363,Z 1139.236,A -85,B 0,C 180,E1 9827.631,E2 9827.631} C_VEL
LIN {X 0,Y 197.148,Z 1143.868,A -85,B 0,C 180,E1 9821.408,E2 9821.408} C_VEL
LIN {X 0,Y 194.217,Z 1147.946,A -85,B 0,C 180,E1 9813.837,E2 9813.837} C_VEL
LIN {X 0,Y 193.15,Z 1150.192,A -85,B 0,C 180,E1 9807.033,E2 9807.033} C_VEL
LIN {X 0,Y 192.973,Z 1151.255,A -85,B 0,C 180,E1 9801.358,E2 9801.358} C_VEL
LIN {X 0,Y 193.209,Z 1151.567,A -85,B 0,C 180,E1 9795.617,E2 9795.617} C_VEL
LIN {X 0,Y 194.157,Z 1151.046,A -85,B 0,C 180,E1 9789.501,E2 9789.501} C_VEL
LIN {X 0,Y 196.253,Z 1149.614,A -85,B 0,C 180,E1 9783.363,E2 9783.363} C_VEL
LIN {X 0,Y 199.968,Z 1147.153,A -85,B 0,C 180,E1 9777.145,E2 9777.145} C_VEL
LIN {X 0,Y 206.97,Z 1142.755,A -85,B 0,C 180,E1 9769.757,E2 9769.757} C_VEL
LIN {X 0,Y 216.71,Z 1136.441,A -85,B 0,C 180,E1 9762.811,E2 9762.811} C_VEL
LIN {X 0,Y 226.276,Z 1130.242,A -85,B 0,C 180,E1 9757.725,E2 9757.725} C_VEL
LIN {X 0,Y 239.255,Z 1121.624,A -85,B 0,C 180,E1 9752.34,E2 9752.34} C_VEL
LIN {X 0,Y 254.43,Z 1110.79,A -85,B 0,C 180,E1 9747.36,E2 9747.36} C_VEL
LIN {X 0,Y 267.763,Z 1100.724,A -85,B 0,C 180,E1 9743.785,E2 9743.785} C_VEL
LIN {X 0,Y 281.956,Z 1089.33,A -85,B 0,C 180,E1 9740.554,E2 9740.554} C_VEL
LIN {X 0,Y 300.19,Z 1073.424,A -85,B 0,C 180,E1 9737.045,E2 9737.045} C_VEL
LIN {X 0,Y 314.264,Z 1060.005,A -85,B 0,C 180,E1 9734.715,E2 9734.715} C_VEL
LIN {X 0,Y 328.188,Z 1045.672,A -85,B 0,C 180,E1 9732.672,E2 9732.672} C_VEL
LIN {X 0,Y 343.851,Z 1028.152,A -85,B 0,C 180,E1 9730.628,E2 9730.628} C_VEL
LIN {X 0,Y 359.434,Z 1008.585,A -85,B 0,C 180,E1 9728.801,E2 9728.801} C_VEL
LIN {X 0,Y 371.628,Z 991.717,A -85,B 0,C 180,E1 9727.501,E2 9727.501} C_VEL
LIN {X 0,Y 383.293,Z 973.971,A -85,B 0,C 180,E1 9726.344,E2 9726.344} C_VEL
LIN {X 0,Y 396.533,Z 951.528,A -85,B 0,C 180,E1 9725.13,E2 9725.13} C_VEL
LIN {X 0,Y 408.009,Z 928.942,A -85,B 0,C 180,E1 9724.144,E2 9724.144} C_VEL
LIN {X 0,Y 416.688,Z 909.575,A -85,B 0,C 180,E1 9723.432,E2 9723.432} C_VEL
LIN {X 0,Y 425.183,Z 887.854,A -85,B 0,C 180,E1 9722.76,E2 9722.76} C_VEL
LIN {X 0,Y 434.082,Z 860.251,A -85,B 0,C 180,E1 9722.08,E2 9722.08} C_VEL
LIN {X 0,Y 439.608,Z 838.945,A -85,B 0,C 180,E1 9721.667,E2 9721.667} C_VEL
LIN {X 0,Y 444.142,Z 817.036,A -85,B 0,C 180,E1 9721.317,E2 9721.317} C_VEL
LIN {X 0,Y 448.341,Z 788.996,A -85,B 0,C 180,E1 9720.947,E2 9720.947} C_VEL
LIN {X 0,Y 463.72,Z 659.833,A -85,B 0,C 180,E1 9719.331,E2 9719.331} C_VEL
LIN {X 0,Y 464.02,Z 657.165,A -85,B 0,C 180,E1 9719.197,E2 9719.197} C_VEL
LIN {X 0,Y 464.768,Z 650.094,A -85,B 0,C 180,E1 9718.318,E2 9718.318} C_VEL
LIN {X 0,Y 465.088,Z 647.427,A -85,B 0,C 180,E1 9718.187,E2 9718.187} C_VEL
LIN {X 0,Y 465.554,Z 643.618,A -85,B 0,C 180,E1 9718.123,E2 9718.123} C_VEL
LIN {X 0,Y 465.541,Z 644.143,A -85,B 0,C 180,E1 9716.899,E2 9716.899} C_VEL
LIN {X 0,Y 445.904,Z 805.425,A -85,B 0,C 180,E1 9714.832,E2 9714.832} C_VEL
LIN {X 0,Y 441.092,Z 832.71,A -85,B 0,C 180,E1 9714.459,E2 9714.459} C_VEL
LIN {X 0,Y 434.693,Z 858.555,A -85,B 0,C 180,E1 9714.074,E2 9714.074} C_VEL
LIN {X 0,Y 428.274,Z 879.729,A -85,B 0,C 180,E1 9713.71,E2 9713.71} C_VEL
LIN {X 0,Y 420.368,Z 901.86,A -85,B 0,C 180,E1 9713.234,E2 9713.234} C_VEL
LIN {X 0,Y 408.946,Z 928.737,A -85,B 0,C 180,E1 9712.495,E2 9712.495} C_VEL
LIN {X 0,Y 398.73,Z 949.463,A -85,B 0,C 180,E1 9711.782,E2 9711.782} C_VEL
LIN {X 0,Y 388.238,Z 968.507,A -85,B 0,C 180,E1 9710.989,E2 9710.989} C_VEL
LIN {X 0,Y 374.468,Z 990.985,A -85,B 0,C 180,E1 9709.85,E2 9709.85} C_VEL
LIN {X 0,Y 358.97,Z 1013.191,A -85,B 0,C 180,E1 9708.431,E2 9708.431} C_VEL
LIN {X 0,Y 346.509,Z 1029.496,A -85,B 0,C 180,E1 9707.162,E2 9707.162} C_VEL
LIN {X 0,Y 332.425,Z 1046.485,A -85,B 0,C 180,E1 9705.581,E2 9705.581} C_VEL
LIN {X 0,Y 315.144,Z 1065.729,A -85,B 0,C 180,E1 9703.367,E2 9703.367} C_VEL
LIN {X 0,Y 297.584,Z 1083.379,A -85,B 0,C 180,E1 9700.759,E2 9700.759} C_VEL
LIN {X 0,Y 282.879,Z 1097.206,A -85,B 0,C 180,E1 9698.214,E2 9698.214} C_VEL
LIN {X 0,Y 267.739,Z 1110.624,A -85,B 0,C 180,E1 9695.159,E2 9695.159} C_VEL
LIN {X 0,Y 248.423,Z 1126.711,A -85,B 0,C 180,E1 9690.385,E2 9690.385} C_VEL
LIN {X 0,Y 234.723,Z 1137.571,A -85,B 0,C 180,E1 9686.166,E2 9686.166} C_VEL
LIN {X 0,Y 222.389,Z 1147.145,A -85,B 0,C 180,E1 9681.472,E2 9681.472} C_VEL
LIN {X 0,Y 209.27,Z 1157.398,A -85,B 0,C 180,E1 9674.997,E2 9674.997} C_VEL
LIN {X 0,Y 198.855,Z 1165.661,A -85,B 0,C 180,E1 9667.838,E2 9667.838} C_VEL
LIN {X 0,Y 192.323,Z 1171.401,A -85,B 0,C 180,E1 9661.325,E2 9661.325} C_VEL
LIN {X 0,Y 188.049,Z 1175.778,A -85,B 0,C 180,E1 9654.838,E2 9654.838} C_VEL
LIN {X 0,Y 185.511,Z 1179.218,A -85,B 0,C 180,E1 9647.892,E2 9647.892} C_VEL
LIN {X 0,Y 184.627,Z 1181.386,A -85,B 0,C 180,E1 9641.243,E2 9641.243} C_VEL
LIN {X 0,Y 184.686,Z 1182.363,A -85,B 0,C 180,E1 9635.281,E2 9635.281} C_VEL
LIN {X 0,Y 184.831,Z 1182.414,A -85,B 0,C 180,E1 9630.31,E2 9630.31} C_VEL
LIN {X 0,Y 184.765,Z 1181.835,A -85,B 0,C 180,E1 9625.655,E2 9625.655} C_VEL
LIN {X 0,Y 184.686,Z 1180.285,A -85,B 0,C 180,E1 9620.024,E2 9620.024} C_VEL
LIN {X 0,Y 185.333,Z 1177.309,A -85,B 0,C 180,E1 9613.386,E2 9613.386} C_VEL
LIN {X 0,Y 187.349,Z 1173.138,A -85,B 0,C 180,E1 9606.739,E2 9606.739} C_VEL
LIN {X 0,Y 190.857,Z 1168.047,A -85,B 0,C 180,E1 9600.499,E2 9600.499} C_VEL
LIN {X 0,Y 196.069,Z 1161.835,A -85,B 0,C 180,E1 9594.455,E2 9594.455} C_VEL
LIN {X 0,Y 204.169,Z 1153.298,A -85,B 0,C 180,E1 9587.862,E2 9587.862} C_VEL
LIN {X 0,Y 215.499,Z 1142.007,A -85,B 0,C 180,E1 9581.214,E2 9581.214} C_VEL
LIN {X 0,Y 226.152,Z 1131.621,A -85,B 0,C 180,E1 9576.424,E2 9576.424} C_VEL
LIN {X 0,Y 237.579,Z 1120.386,A -85,B 0,C 180,E1 9572.23,E2 9572.23} C_VEL
LIN {X 0,Y 252.147,Z 1105.726,A -85,B 0,C 180,E1 9567.837,E2 9567.837} C_VEL
LIN {X 0,Y 267.292,Z 1089.463,A -85,B 0,C 180,E1 9564.064,E2 9564.064} C_VEL
LIN {X 0,Y 280.166,Z 1074.921,A -85,B 0,C 180,E1 9561.337,E2 9561.337} C_VEL
LIN {X 0,Y 293.36,Z 1059.111,A -85,B 0,C 180,E1 9558.893,E2 9558.893} C_VEL
LIN {X 0,Y 309.391,Z 1038.344,A -85,B 0,C 180,E1 9556.299,E2 9556.299} C_VEL
LIN {X 0,Y 322.609,Z 1019.492,A -85,B 0,C 180,E1 9554.414,E2 9554.414} C_VEL
LIN {X 0,Y 333.94,Z 1001.944,A -85,B 0,C 180,E1 9552.946,E2 9552.946} C_VEL
LIN {X 0,Y 346.314,Z 981.028,A -85,B 0,C 180,E1 9551.491,E2 9551.491} C_VEL
LIN {X 0,Y 359.089,Z 956.616,A -85,B 0,C 180,E1 9550.124,E2 9550.124} C_VEL
LIN {X 0,Y 368.669,Z 935.932,A -85,B 0,C 180,E1 9549.18,E2 9549.18} C_VEL
LIN {X 0,Y 377.431,Z 914.621,A -85,B 0,C 180,E1 9548.378,E2 9548.378} C_VEL
LIN {X 0,Y 386.781,Z 888.127,A -85,B 0,C 180,E1 9547.576,E2 9547.576} C_VEL
LIN {X 0,Y 393.678,Z 864.349,A -85,B 0,C 180,E1 9547.022,E2 9547.022} C_VEL
LIN {X 0,Y 398.951,Z 842.247,A -85,B 0,C 180,E1 9546.603,E2 9546.603} C_VEL
LIN {X 0,Y 403.88,Z 815.334,A -85,B 0,C 180,E1 9546.147,E2 9546.147} C_VEL
LIN {X 0,Y 409.088,Z 769.412,A -85,B 0,C 180,E1 9545.484,E2 9545.484} C_VEL
LIN {X 0,Y 425.911,Z 610.16,A -85,B 0,C 180,E1 9543.248,E2 9543.248} C_VEL
LIN {X 0,Y 423.806,Z 604.697,A -85,B 0,C 180,E1 9540.879,E2 9540.879} C_VEL
LIN {X 0,Y 422.545,Z 601.67,A -85,B 0,C 180,E1 9539.051,E2 9539.051} C_VEL
LIN {X 0,Y 421.491,Z 598.874,A -85,B 0,C 180,E1 9536.872,E2 9536.872} C_VEL
LIN {X 0,Y 420.709,Z 596.97,A -85,B 0,C 180,E1 9533.038,E2 9533.038} C_VEL
LIN {X 0,Y 421.108,Z 598.149,A -85,B 0,C 180,E1 9529.88,E2 9529.88} C_VEL
LIN {X 0,Y 421.793,Z 599.536,A -85,B 0,C 180,E1 9528.098,E2 9528.098} C_VEL
LIN {X 0,Y 423.315,Z 603.35,A -85,B 0,C 180,E1 9525.5,E2 9525.5} C_VEL
LIN {X 0,Y 424.747,Z 606.946,A -85,B 0,C 180,E1 9523.702,E2 9523.702} C_VEL
LIN {X 0,Y 403.712,Z 800.317,A -85,B 0,C 180,E1 9521.087,E2 9521.087} C_VEL
LIN {X 0,Y 399.4,Z 826.986,A -85,B 0,C 180,E1 9520.655,E2 9520.655} C_VEL
LIN {X 0,Y 393.686,Z 851.989,A -85,B 0,C 180,E1 9520.13,E2 9520.13} C_VEL
LIN {X 0,Y 387.823,Z 872.964,A -85,B 0,C 180,E1 9519.578,E2 9519.578} C_VEL
LIN {X 0,Y 380.551,Z 895.001,A -85,B 0,C 180,E1 9518.863,E2 9518.863} C_VEL
LIN {X 0,Y 370.332,Z 920.919,A -85,B 0,C 180,E1 9517.829,E2 9517.829} C_VEL
LIN {X 0,Y 361.039,Z 941.213,A -85,B 0,C 180,E1 9516.844,E2 9516.844} C_VEL
LIN {X 0,Y 351.016,Z 960.733,A -85,B 0,C 180,E1 9515.714,E2 9515.714} C_VEL
LIN {X 0,Y 337.447,Z 984.152,A -85,B 0,C 180,E1 9514.062,E2 9514.062} C_VEL
LIN {X 0,Y 325.34,Z 1002.705,A -85,B 0,C 180,E1 9512.453,E2 9512.453} C_VEL
LIN {X 0,Y 313.875,Z 1018.806,A -85,B 0,C 180,E1 9510.789,E2 9510.789} C_VEL
LIN {X 0,Y 300.004,Z 1036.744,A -85,B 0,C 180,E1 9508.561,E2 9508.561} C_VEL
LIN {X 0,Y 285.098,Z 1054.169,A -85,B 0,C 180,E1 9505.86,E2 9505.86} C_VEL
LIN {X 0,Y 272.228,Z 1068.119,A -85,B 0,C 180,E1 9503.195,E2 9503.195} C_VEL
LIN {X 0,Y 259.944,Z 1080.631,A -85,B 0,C 180,E1 9500.29,E2 9500.29} C_VEL
LIN {X 0,Y 245.232,Z 1094.811,A -85,B 0,C 180,E1 9496.192,E2 9496.192} C_VEL
LIN {X 0,Y 231.741,Z 1106.9,A -85,B 0,C 180,E1 9491.639,E2 9491.639} C_VEL
LIN {X 0,Y 220.692,Z 1116.53,A -85,B 0,C 180,E1 9487.053,E2 9487.053} C_VEL
LIN {X 0,Y 209.312,Z 1126.387,A -85,B 0,C 180,E1 9481.058,E2 9481.058} C_VEL
LIN {X 0,Y 200.044,Z 1134.331,A -85,B 0,C 180,E1 9474.51,E2 9474.51} C_VEL
LIN {X 0,Y 193.786,Z 1140.078,A -85,B 0,C 180,E1 9468.345,E2 9468.345} C_VEL
LIN {X 0,Y 189.036,Z 1145.061,A -85,B 0,C 180,E1 9461.285,E2 9461.285} C_VEL
LIN {X 0,Y 186.124,Z 1148.895,A -85,B 0,C 180,E1 9453.387,E2 9453.387} C_VEL
LIN {X 0,Y 185.165,Z 1150.9,A -85,B 0,C 180,E1 9446.904,E2 9446.904} C_VEL
LIN {X 0,Y 184.999,Z 1151.908,A -85,B 0,C 180,E1 9441.296,E2 9441.296} C_VEL
LIN {X 0,Y 185.261,Z 1152.236,A -85,B 0,C 180,E1 9435.306,E2 9435.306} C_VEL
LIN {X 0,Y 186.312,Z 1151.731,A -85,B 0,C 180,E1 9428.927,E2 9428.927} C_VEL
LIN {X 0,Y 188.61,Z 1150.317,A -85,B 0,C 180,E1 9422.535,E2 9422.535} C_VEL
LIN {X 0,Y 192.565,Z 1147.917,A -85,B 0,C 180,E1 9416.181,E2 9416.181} C_VEL
LIN {X 0,Y 199.544,Z 1143.821,A -85,B 0,C 180,E1 9408.974,E2 9408.974} C_VEL
LIN {X 0,Y 210.035,Z 1137.499,A -85,B 0,C 180,E1 9401.635,E2 9401.635} C_VEL
LIN {X 0,Y 220.565,Z 1131.033,A -85,B 0,C 180,E1 9396.205,E2 9396.205} C_VEL
LIN {X 0,Y 233.4,Z 1122.89,A -85,B 0,C 180,E1 9391.043,E2 9391.043} C_VEL
LIN {X 0,Y 249.896,Z 1111.64,A -85,B 0,C 180,E1 9385.809,E2 9385.809} C_VEL
LIN {X 0,Y 263.629,Z 1101.628,A -85,B 0,C 180,E1 9382.269,E2 9382.269} C_VEL
LIN {X 0,Y 278.24,Z 1090.265,A -85,B 0,C 180,E1 9379.075,E2 9379.075} C_VEL
LIN {X 0,Y 296.934,Z 1074.429,A -85,B 0,C 180,E1 9375.626,E2 9375.626} C_VEL
LIN {X 0,Y 312.217,Z 1060.168,A -85,B 0,C 180,E1 9373.209,E2 9373.209} C_VEL
LIN {X 0,Y 326.668,Z 1045.55,A -85,B 0,C 180,E1 9371.192,E2 9371.192} C_VEL
LIN {X 0,Y 343.306,Z 1027.146,A -85,B 0,C 180,E1 9369.135,E2 9369.135} C_VEL
LIN {X 0,Y 358.475,Z 1008.25,A -85,B 0,C 180,E1 9367.449,E2 9367.449} C_VEL
LIN {X 0,Y 370.678,Z 991.576,A -85,B 0,C 180,E1 9366.217,E2 9366.217} C_VEL
LIN {X 0,Y 382.893,Z 973.184,A -85,B 0,C 180,E1 9365.067,E2 9365.067} C_VEL
LIN {X 0,Y 397.322,Z 948.526,A -85,B 0,C 180,E1 9363.809,E2 9363.809} C_VEL
LIN {X 0,Y 407.495,Z 928.584,A -85,B 0,C 180,E1 9362.984,E2 9362.984} C_VEL
LIN {X 0,Y 416.277,Z 909.112,A -85,B 0,C 180,E1 9362.3,E2 9362.3} C_VEL
LIN {X 0,Y 425.852,Z 884.656,A -85,B 0,C 180,E1 9361.583,E2 9361.583} C_VEL
LIN {X 0,Y 433.968,Z 858.91,A -85,B 0,C 180,E1 9360.987,E2 9360.987} C_VEL
LIN {X 0,Y 439.337,Z 838.174,A -85,B 0,C 180,E1 9360.606,E2 9360.606} C_VEL
LIN {X 0,Y 444.003,Z 815.533,A -85,B 0,C 180,E1 9360.261,E2 9360.261} C_VEL
LIN {X 0,Y 448.954,Z 780.55,A -85,B 0,C 180,E1 9359.816,E2 9359.816} C_VEL
LIN {X 0,Y 465.088,Z 647.427,A -85,B 0,C 180,E1 9358.187,E2 9358.187} C_VEL
LIN {X 0,Y 464.912,Z 648.794,A -85,B 0,C 180,E1 9358.044,E2 9358.044} C_VEL
LIN {X 0,Y 463.888,Z 657.051,A -85,B 0,C 180,E1 9357.811,E2 9357.811} C_VEL
LIN {X 0,Y 461.436,Z 676.949,A -85,B 0,C 180,E1 9357.618,E2 9357.618} C_VEL
LIN {X 0,Y 460.319,Z 685.998,A -85,B 0,C 180,E1 9357.655,E2 9357.655} C_VEL
LIN {X 0,Y 445.562,Z 804.333,A -85,B 0,C 180,E1 9359.082,E2 9359.082} C_VEL
LIN {X 0,Y 440.614,Z 831.507,A -85,B 0,C 180,E1 9359.45,E2 9359.45} C_VEL
LIN {X 0,Y 434.48,Z 855.922,A -85,B 0,C 180,E1 9359.861,E2 9359.861} C_VEL
LIN {X 0,Y 427.946,Z 877.194,A -85,B 0,C 180,E1 9360.32,E2 9360.32} C_VEL
LIN {X 0,Y 419.99,Z 899.063,A -85,B 0,C 180,E1 9360.883,E2 9360.883} C_VEL
LIN {X 0,Y 409.012,Z 924.371,A -85,B 0,C 180,E1 9361.681,E2 9361.681} C_VEL
LIN {X 0,Y 398.812,Z 944.614,A -85,B 0,C 180,E1 9362.462,E2 9362.462} C_VEL
LIN {X 0,Y 388.586,Z 962.707,A -85,B 0,C 180,E1 9363.292,E2 9363.292} C_VEL
LIN {X 0,Y 375.082,Z 984.102,A -85,B 0,C 180,E1 9364.459,E2 9364.459} C_VEL
LIN {X 0,Y 359.844,Z 1005.188,A -85,B 0,C 180,E1 9365.883,E2 9365.883} C_VEL
LIN {X 0,Y 346.711,Z 1021.607,A -85,B 0,C 180,E1 9367.233,E2 9367.233} C_VEL
LIN {X 0,Y 332.691,Z 1037.627,A -85,B 0,C 180,E1 9368.817,E2 9368.817} C_VEL
LIN {X 0,Y 314.826,Z 1056.123,A -85,B 0,C 180,E1 9371.081,E2 9371.081} C_VEL
LIN {X 0,Y 299.051,Z 1070.811,A -85,B 0,C 180,E1 9373.359,E2 9373.359} C_VEL
LIN {X 0,Y 284.623,Z 1083.211,A -85,B 0,C 180,E1 9375.732,E2 9375.732} C_VEL
LIN {X 0,Y 269.132,Z 1095.55,A -85,B 0,C 180,E1 9378.674,E2 9378.674} C_VEL
LIN {X 0,Y 250.673,Z 1108.979,A -85,B 0,C 180,E1 9382.87,E2 9382.87} C_VEL
LIN {X 0,Y 236.414,Z 1118.55,A -85,B 0,C 180,E1 9386.827,E2 9386.827} C_VEL
LIN {X 0,Y 223.145,Z 1126.946,A -85,B 0,C 180,E1 9391.318,E2 9391.318} C_VEL
LIN {X 0,Y 208.479,Z 1135.709,A -85,B 0,C 180,E1 9397.689,E2 9397.689} C_VEL
LIN {X 0,Y 197.558,Z 1141.851,A -85,B 0,C 180,E1 9404.055,E2 9404.055} C_VEL
LIN {X 0,Y 189.651,Z 1146.246,A -85,B 0,C 180,E1 9410.363,E2 9410.363} C_VEL
LIN {X 0,Y 182.761,Z 1150.141,A -85,B 0,C 180,E1 9418.593,E2 9418.593} C_VEL
LIN {X 0,Y 178.967,Z 1152.158,A -85,B 0,C 180,E1 9426.63,E2 9426.63} C_VEL
LIN {X 0,Y 177.547,Z 1152.84,A -85,B 0,C 180,E1 9432.972,E2 9432.972} C_VEL
LIN {X 0,Y 177.057,Z 1152.763,A -85,B 0,C 180,E1 9438.93,E2 9438.93} C_VEL
LIN {X 0,Y 177.081,Z 1152.013,A -85,B 0,C 180,E1 9444.817,E2 9444.817} C_VEL
LIN {X 0,Y 177.721,Z 1150.381,A -85,B 0,C 180,E1 9451.289,E2 9451.289} C_VEL
LIN {X 0,Y 179.416,Z 1147.896,A -85,B 0,C 180,E1 9457.686,E2 9457.686} C_VEL
LIN {X 0,Y 182.655,Z 1144.328,A -85,B 0,C 180,E1 9464.26,E2 9464.26} C_VEL
LIN {X 0,Y 188.137,Z 1139.264,A -85,B 0,C 180,E1 9471.185,E2 9471.185} C_VEL
LIN {X 0,Y 197.583,Z 1131.279,A -85,B 0,C 180,E1 9479.065,E2 9479.065} C_VEL
LIN {X 0,Y 207.017,Z 1123.55,A -85,B 0,C 180,E1 9484.744,E2 9484.744} C_VEL
LIN {X 0,Y 218.074,Z 1114.503,A -85,B 0,C 180,E1 9489.933,E2 9489.933} C_VEL
LIN {X 0,Y 232.969,Z 1101.863,A -85,B 0,C 180,E1 9495.434,E2 9495.434} C_VEL
LIN {X 0,Y 245.585,Z 1090.57,A -85,B 0,C 180,E1 9499.224,E2 9499.224} C_VEL
LIN {X 0,Y 258.388,Z 1078.497,A -85,B 0,C 180,E1 9502.492,E2 9502.492} C_VEL
LIN {X 0,Y 274.086,Z 1062.732,A -85,B 0,C 180,E1 9505.903,E2 9505.903} C_VEL
LIN {X 0,Y 289.032,Z 1046.183,A -85,B 0,C 180,E1 9508.699,E2 9508.699} C_VEL
LIN {X 0,Y 301.409,Z 1031.427,A -85,B 0,C 180,E1 9510.743,E2 9510.743} C_VEL
LIN {X 0,Y 314.518,Z 1014.503,A -85,B 0,C 180,E1 9512.689,E2 9512.689} C_VEL
LIN {X 0,Y 329.971,Z 992.265,A -85,B 0,C 180,E1 9514.755,E2 9514.755} C_VEL
LIN {X 0,Y 341.176,Z 974.291,A -85,B 0,C 180,E1 9516.114,E2 9516.114} C_VEL
LIN {X 0,Y 351.261,Z 956.456,A -85,B 0,C 180,E1 9517.258,E2 9517.258} C_VEL
LIN {X 0,Y 362.754,Z 933.811,A -85,B 0,C 180,E1 9518.473,E2 9518.473} C_VEL
LIN {X 0,Y 373.054,Z 909.95,A -85,B 0,C 180,E1 9519.509,E2 9519.509} C_VEL
LIN {X 0,Y 380.699,Z 889.631,A -85,B 0,C 180,E1 9520.232,E2 9520.232} C_VEL
LIN {X 0,Y 387.381,Z 869.02,A -85,B 0,C 180,E1 9520.851,E2 9520.851} C_VEL
LIN {X 0,Y 394.741,Z 841.201,A -85,B 0,C 180,E1 9521.519,E2 9521.519} C_VEL
LIN {X 0,Y 399.46,Z 817.847,A -85,B 0,C 180,E1 9521.944,E2 9521.944} C_VEL
LIN {X 0,Y 402.858,Z 795.233,A -85,B 0,C 180,E1 9522.278,E2 9522.278} C_VEL
LIN {X 0,Y 422.901,Z 612.903,A -85,B 0,C 180,E1 9524.714,E2 9524.714} C_VEL
LIN {X 0,Y 421.439,Z 609.327,A -85,B 0,C 180,E1 9526.834,E2 9526.834} C_VEL
LIN {X 0,Y 420.42,Z 606.613,A -85,B 0,C 180,E1 9529.032,E2 9529.032} C_VEL
LIN {X 0,Y 419.73,Z 604.922,A -85,B 0,C 180,E1 9532.747,E2 9532.747} C_VEL
LIN {X 0,Y 420.193,Z 606.315,A -85,B 0,C 180,E1 9536.043,E2 9536.043} C_VEL
LIN {X 0,Y 420.733,Z 607.504,A -85,B 0,C 180,E1 9537.438,E2 9537.438} C_VEL
LIN {X 0,Y 422.196,Z 611.368,A -85,B 0,C 180,E1 9540.068,E2 9540.068} C_VEL
LIN {X 0,Y 423.937,Z 616.033,A -85,B 0,C 180,E1 9542.273,E2 9542.273} C_VEL
LIN {X 0,Y 403.146,Z 807.639,A -85,B 0,C 180,E1 9544.92,E2 9544.92} C_VEL
LIN {X 0,Y 398.763,Z 834.8,A -85,B 0,C 180,E1 9545.349,E2 9545.349} C_VEL
LIN {X 0,Y 392.69,Z 860.921,A -85,B 0,C 180,E1 9545.816,E2 9545.816} C_VEL
LIN {X 0,Y 386.755,Z 881.746,A -85,B 0,C 180,E1 9546.266,E2 9546.266} C_VEL
LIN {X 0,Y 379.407,Z 903.699,A -85,B 0,C 180,E1 9546.854,E2 9546.854} C_VEL
LIN {X 0,Y 368.777,Z 930.562,A -85,B 0,C 180,E1 9547.764,E2 9547.764} C_VEL
LIN {X 0,Y 359.043,Z 951.736,A -85,B 0,C 180,E1 9548.661,E2 9548.661} C_VEL
LIN {X 0,Y 349.238,Z 970.852,A -85,B 0,C 180,E1 9549.635,E2 9549.635} C_VEL
LIN {X 0,Y 337.22,Z 992.046,A -85,B 0,C 180,E1 9550.939,E2 9550.939} C_VEL
LIN {X 0,Y 322.794,Z 1014.627,A -85,B 0,C 180,E1 9552.653,E2 9552.653} C_VEL
LIN {X 0,Y 310.108,Z 1032.662,A -85,B 0,C 180,E1 9554.332,E2 9554.332} C_VEL
LIN {X 0,Y 297.458,Z 1049.3,A -85,B 0,C 180,E1 9556.201,E2 9556.201} C_VEL
LIN {X 0,Y 281.706,Z 1068.506,A -85,B 0,C 180,E1 9558.844,E2 9558.844} C_VEL
LIN {X 0,Y 266.136,Z 1085.81,A -85,B 0,C 180,E1 9561.881,E2 9561.881} C_VEL
LIN {X 0,Y 253.318,Z 1099.281,A -85,B 0,C 180,E1 9564.795,E2 9564.795} C_VEL
LIN {X 0,Y 239.815,Z 1112.811,A -85,B 0,C 180,E1 9568.392,E2 9568.392} C_VEL
LIN {X 0,Y 223.582,Z 1128.334,A -85,B 0,C 180,E1 9573.717,E2 9573.717} C_VEL
LIN {X 0,Y 212.011,Z 1139.104,A -85,B 0,C 180,E1 9578.502,E2 9578.502} C_VEL
LIN {X 0,Y 201.95,Z 1148.49,A -85,B 0,C 180,E1 9583.71,E2 9583.71} C_VEL
LIN {X 0,Y 192.011,Z 1158.212,A -85,B 0,C 180,E1 9590.559,E2 9590.559} C_VEL
LIN {X 0,Y 184.173,Z 1166.545,A -85,B 0,C 180,E1 9598.47,E2 9598.47} C_VEL
LIN {X 0,Y 180.052,Z 1171.872,A -85,B 0,C 180,E1 9605.037,E2 9605.037} C_VEL
LIN {X 0,Y 177.692,Z 1176.003,A -85,B 0,C 180,E1 9611.633,E2 9611.633} C_VEL
LIN {X 0,Y 176.801,Z 1178.79,A -85,B 0,C 180,E1 9617.591,E2 9617.591} C_VEL
LIN {X 0,Y 176.733,Z 1180.62,A -85,B 0,C 180,E1 9623.177,E2 9623.177} C_VEL
LIN {X 0,Y 176.856,Z 1181.645,A -85,B 0,C 180,E1 9628.704,E2 9628.704} C_VEL
LIN {X 0,Y 176.745,Z 1181.852,A -85,B 0,C 180,E1 9634.218,E2 9634.218} C_VEL
LIN {X 0,Y 176.622,Z 1181.1,A -85,B 0,C 180,E1 9640.437,E2 9640.437} C_VEL
LIN {X 0,Y 177.61,Z 1178.736,A -85,B 0,C 180,E1 9648.376,E2 9648.376} C_VEL
LIN {X 0,Y 180.351,Z 1175.362,A -85,B 0,C 180,E1 9655.622,E2 9655.622} C_VEL
LIN {X 0,Y 185.201,Z 1170.82,A -85,B 0,C 180,E1 9662.675,E2 9662.675} C_VEL
LIN {X 0,Y 192.251,Z 1165.103,A -85,B 0,C 180,E1 9669.383,E2 9669.383} C_VEL
LIN {X 0,Y 203.358,Z 1156.87,A -85,B 0,C 180,E1 9676.692,E2 9676.692} C_VEL
LIN {X 0,Y 217.263,Z 1146.619,A -85,B 0,C 180,E1 9683.252,E2 9683.252} C_VEL
LIN {X 0,Y 230.429,Z 1136.871,A -85,B 0,C 180,E1 9688.036,E2 9688.036} C_VEL
LIN {X 0,Y 245.754,Z 1125.216,A -85,B 0,C 180,E1 9692.492,E2 9692.492} C_VEL
LIN {X 0,Y 264.403,Z 1110.192,A -85,B 0,C 180,E1 9696.84,E2 9696.84} C_VEL
LIN {X 0,Y 280.1,Z 1096.685,A -85,B 0,C 180,E1 9699.854,E2 9699.854} C_VEL
LIN {X 0,Y 294.926,Z 1083.098,A -85,B 0,C 180,E1 9702.297,E2 9702.297} C_VEL
LIN {X 0,Y 312.857,Z 1065.485,A -85,B 0,C 180,E1 9704.832,E2 9704.832} C_VEL
LIN {X 0,Y 330.904,Z 1045.818,A -85,B 0,C 180,E1 9707.024,E2 9707.024} C_VEL
LIN {X 0,Y 344.864,Z 1029.276,A -85,B 0,C 180,E1 9708.509,E2 9708.509} C_VEL
LIN {X 0,Y 358.117,Z 1012.204,A -85,B 0,C 180,E1 9709.782,E2 9709.782} C_VEL
LIN {X 0,Y 373.734,Z 990.059,A -85,B 0,C 180,E1 9711.134,E2 9711.134} C_VEL
LIN {X 0,Y 387.05,Z 968.615,A -85,B 0,C 180,E1 9712.175,E2 9712.175} C_VEL
LIN {X 0,Y 397.949,Z 949.083,A -85,B 0,C 180,E1 9712.955,E2 9712.955} C_VEL
LIN {X 0,Y 407.973,Z 928.99,A -85,B 0,C 180,E1 9713.616,E2 9713.616} C_VEL
LIN {X 0,Y 419.02,Z 903.609,A -85,B 0,C 180,E1 9714.29,E2 9714.29} C_VEL
LIN {X 0,Y 427.71,Z 879.656,A -85,B 0,C 180,E1 9714.786,E2 9714.786} C_VEL
LIN {X 0,Y 434.329,Z 858.037,A -85,B 0,C 180,E1 9715.139,E2 9715.139} C_VEL
LIN {X 0,Y 440.881,Z 831.747,A -85,B 0,C 180,E1 9715.516,E2 9715.516} C_VEL
LIN {X 0,Y 445.649,Z 804.779,A -85,B 0,C 180,E1 9715.872,E2 9715.872} C_VEL
LIN {X 0,Y 461.762,Z 674.327,A -85,B 0,C 180,E1 9717.516,E2 9717.516} C_VEL
LIN {X 0,Y 460.319,Z 685.998,A -85,B 0,C 180,E1 9717.655,E2 9717.655} C_VEL
LIN {X 0,Y 460.301,Z 686.298,A -85,B 0,C 180,E1 9717.657,E2 9717.657} C_VEL
LIN {X 0,Y 460.301,Z 822.824,A -85,B 0,C 180,E1 9717.657,E2 9717.657} C_VEL
LIN {X 0,Y 454.318,Z 822.824,A -85,B 0,C 180,E1 9717.884,E2 9717.884} C_VEL
LIN {X 0,Y 452.405,Z 820.824,A -85,B 0,C 180,E1 9717.958,E2 9717.958} C_VEL
LIN {X 0,Y 452.405,Z 758.416,A -85,B 0,C 180,E1 9717.958,E2 9717.958} C_VEL
LIN {X 0,Y 451.505,Z 757.499,A -85,B 0,C 180,E1 9717.493,E2 9717.493} C_VEL
LIN {X 0,Y 444.857,Z 808.854,A -85,B 0,C 180,E1 9716.854,E2 9716.854} C_VEL
LIN {X 0,Y 439.322,Z 837.105,A -85,B 0,C 180,E1 9716.488,E2 9716.488} C_VEL
LIN {X 0,Y 433.529,Z 859.579,A -85,B 0,C 180,E1 9716.177,E2 9716.177} C_VEL
LIN {X 0,Y 426.739,Z 881.28,A -85,B 0,C 180,E1 9715.835,E2 9715.835} C_VEL
LIN {X 0,Y 416.842,Z 907.599,A -85,B 0,C 180,E1 9715.301,E2 9715.301} C_VEL
LIN {X 0,Y 406.674,Z 930.281,A -85,B 0,C 180,E1 9714.712,E2 9714.712} C_VEL
LIN {X 0,Y 397.039,Z 949.269,A -85,B 0,C 180,E1 9714.111,E2 9714.111} C_VEL
LIN {X 0,Y 385.552,Z 969.534,A -85,B 0,C 180,E1 9713.334,E2 9713.334} C_VEL
LIN {X 0,Y 369.899,Z 993.92,A -85,B 0,C 180,E1 9712.168,E2 9712.168} C_VEL
LIN {X 0,Y 355.832,Z 1013.356,A -85,B 0,C 180,E1 9710.999,E2 9710.999} C_VEL
LIN {X 0,Y 342.396,Z 1030.294,A -85,B 0,C 180,E1 9709.769,E2 9709.769} C_VEL
LIN {X 0,Y 325.508,Z 1049.799,A -85,B 0,C 180,E1 9708.031,E2 9708.031} C_VEL
LIN {X 0,Y 307.234,Z 1068.708,A -85,B 0,C 180,E1 9705.872,E2 9705.872} C_VEL
LIN {X 0,Y 291.63,Z 1083.606,A -85,B 0,C 180,E1 9703.737,E2 9703.737} C_VEL
LIN {X 0,Y 275.66,Z 1097.811,A -85,B 0,C 180,E1 9701.206,E2 9701.206} C_VEL
LIN {X 0,Y 255.591,Z 1114.321,A -85,B 0,C 180,E1 9697.402,E2 9697.402} C_VEL
LIN {X 0,Y 239.025,Z 1126.961,A -85,B 0,C 180,E1 9693.531,E2 9693.531} C_VEL
LIN {X 0,Y 224.351,Z 1137.643,A -85,B 0,C 180,E1 9689.332,E2 9689.332} C_VEL
LIN {X 0,Y 208.044,Z 1149.169,A -85,B 0,C 180,E1 9683.379,E2 9683.379} C_VEL
LIN {X 0,Y 194.167,Z 1158.653,A -85,B 0,C 180,E1 9676.559,E2 9676.559} C_VEL
LIN {X 0,Y 184.623,Z 1165.392,A -85,B 0,C 180,E1 9670.126,E2 9670.126} C_VEL
LIN {X 0,Y 176.867,Z 1171.331,A -85,B 0,C 180,E1 9662.61,E2 9662.61} C_VEL
LIN {X 0,Y 171.062,Z 1176.599,A -85,B 0,C 180,E1 9653.055,E2 9653.055} C_VEL
LIN {X 0,Y 169.028,Z 1179.336,A -85,B 0,C 180,E1 9645.37,E2 9645.37} C_VEL
LIN {X 0,Y 168.636,Z 1180.722,A -85,B 0,C 180,E1 9638.868,E2 9638.868} C_VEL
LIN {X 0,Y 168.814,Z 1181.197,A -85,B 0,C 180,E1 9633.056,E2 9633.056} C_VEL
LIN {X 0,Y 168.861,Z 1180.909,A -85,B 0,C 180,E1 9627.625,E2 9627.625} C_VEL
LIN {X 0,Y 168.716,Z 1179.612,A -85,B 0,C 180,E1 9621.48,E2 9621.48} C_VEL
LIN {X 0,Y 169.301,Z 1176.667,A -85,B 0,C 180,E1 9613.532,E2 9613.532} C_VEL
LIN {X 0,Y 171.716,Z 1172.22,A -85,B 0,C 180,E1 9605.581,E2 9605.581} C_VEL
LIN {X 0,Y 175.933,Z 1166.925,A -85,B 0,C 180,E1 9598.477,E2 9598.477} C_VEL
LIN {X 0,Y 181.868,Z 1160.741,A -85,B 0,C 180,E1 9591.994,E2 9591.994} C_VEL
LIN {X 0,Y 190.535,Z 1152.623,A -85,B 0,C 180,E1 9585.317,E2 9585.317} C_VEL
LIN {X 0,Y 203.45,Z 1141.07,A -85,B 0,C 180,E1 9578.157,E2 9578.157} C_VEL
LIN {X 0,Y 215.159,Z 1130.645,A -85,B 0,C 180,E1 9573.231,E2 9573.231} C_VEL
LIN {X 0,Y 227.508,Z 1119.442,A -85,B 0,C 180,E1 9569.006,E2 9569.006} C_VEL
LIN {X 0,Y 242.364,Z 1105.495,A -85,B 0,C 180,E1 9564.825,E2 9564.825} C_VEL
LIN {X 0,Y 259.1,Z 1088.691,A -85,B 0,C 180,E1 9560.954,E2 9560.954} C_VEL
LIN {X 0,Y 272.74,Z 1074.102,A -85,B 0,C 180,E1 9558.289,E2 9558.289} C_VEL
LIN {X 0,Y 286.483,Z 1058.413,A -85,B 0,C 180,E1 9555.946,E2 9555.946} C_VEL
LIN {X 0,Y 302.842,Z 1038.205,A -85,B 0,C 180,E1 9553.514,E2 9553.514} C_VEL
LIN {X 0,Y 317.187,Z 1018.535,A -85,B 0,C 180,E1 9551.639,E2 9551.639} C_VEL
LIN {X 0,Y 328.727,Z 1001.31,A -85,B 0,C 180,E1 9550.278,E2 9550.278} C_VEL
LIN {X 0,Y 340.637,Z 981.874,A -85,B 0,C 180,E1 9548.992,E2 9548.992} C_VEL
LIN {X 0,Y 354.742,Z 955.918,A -85,B 0,C 180,E1 9547.613,E2 9547.613} C_VEL
LIN {X 0,Y 364.468,Z 935.525,A -85,B 0,C 180,E1 9546.742,E2 9546.742} C_VEL
LIN {X 0,Y 373.01,Z 915.37,A -85,B 0,C 180,E1 9546.03,E2 9546.03} C_VEL
LIN {X 0,Y 382.243,Z 890.39,A -85,B 0,C 180,E1 9545.309,E2 9545.309} C_VEL
LIN {X 0,Y 390.057,Z 864.293,A -85,B 0,C 180,E1 9544.736,E2 9544.736} C_VEL
LIN {X 0,Y 395.466,Z 842.213,A -85,B 0,C 180,E1 9544.345,E2 9544.345} C_VEL
LIN {X 0,Y 400.202,Z 817.306,A -85,B 0,C 180,E1 9543.942,E2 9543.942} C_VEL
LIN {X 0,Y 404.778,Z 780.335,A -85,B 0,C 180,E1 9543.421,E2 9543.421} C_VEL
LIN {X 0,Y 422.056,Z 621.917,A -85,B 0,C 180,E1 9541.259,E2 9541.259} C_VEL
LIN {X 0,Y 420.464,Z 617.577,A -85,B 0,C 180,E1 9538.91,E2 9538.91} C_VEL
LIN {X 0,Y 419.405,Z 614.618,A -85,B 0,C 180,E1 9536.583,E2 9536.583} C_VEL
LIN {X 0,Y 418.752,Z 612.849,A -85,B 0,C 180,E1 9532.867,E2 9532.867} C_VEL
LIN {X 0,Y 419.393,Z 614.507,A -85,B 0,C 180,E1 9529.144,E2 9529.144} C_VEL
LIN {X 0,Y 420.754,Z 618.131,A -85,B 0,C 180,E1 9526.323,E2 9526.323} C_VEL
LIN {X 0,Y 421.133,Z 619.504,A -85,B 0,C 180,E1 9525.693,E2 9525.693} C_VEL
LIN {X 0,Y 400.725,Z 801.124,A -85,B 0,C 180,E1 9523.324,E2 9523.324} C_VEL
LIN {X 0,Y 396.253,Z 827.962,A -85,B 0,C 180,E1 9522.911,E2 9522.911} C_VEL
LIN {X 0,Y 390.43,Z 852.806,A -85,B 0,C 180,E1 9522.42,E2 9522.42} C_VEL
LIN {X 0,Y 384.244,Z 874.343,A -85,B 0,C 180,E1 9521.884,E2 9521.884} C_VEL
LIN {X 0,Y 376.121,Z 898.169,A -85,B 0,C 180,E1 9521.15,E2 9521.15} C_VEL
LIN {X 0,Y 366.057,Z 922.634,A -85,B 0,C 180,E1 9520.215,E2 9520.215} C_VEL
LIN {X 0,Y 356.931,Z 941.988,A -85,B 0,C 180,E1 9519.329,E2 9519.329} C_VEL
LIN {X 0,Y 346.604,Z 961.533,A -85,B 0,C 180,E1 9518.261,E2 9518.261} C_VEL
LIN {X 0,Y 332.75,Z 984.756,A -85,B 0,C 180,E1 9516.714,E2 9516.714} C_VEL
LIN {X 0,Y 320.052,Z 1003.593,A -85,B 0,C 180,E1 9515.167,E2 9515.167} C_VEL
LIN {X 0,Y 308.14,Z 1019.733,A -85,B 0,C 180,E1 9513.581,E2 9513.581} C_VEL
LIN {X 0,Y 293.679,Z 1037.711,A -85,B 0,C 180,E1 9511.448,E2 9511.448} C_VEL
LIN {X 0,Y 277.553,Z 1055.727,A -85,B 0,C 180,E1 9508.751,E2 9508.751} C_VEL
LIN {X 0,Y 264.295,Z 1069.382,A -85,B 0,C 180,E1 9506.211,E2 9506.211} C_VEL
LIN {X 0,Y 250.818,Z 1082.35,A -85,B 0,C 180,E1 9503.251,E2 9503.251} C_VEL
LIN {X 0,Y 234.515,Z 1096.982,A -85,B 0,C 180,E1 9498.994,E2 9498.994} C_VEL
LIN {X 0,Y 220.708,Z 1108.492,A -85,B 0,C 180,E1 9494.602,E2 9494.602} C_VEL
LIN {X 0,Y 209.093,Z 1117.808,A -85,B 0,C 180,E1 9490.081,E2 9490.081} C_VEL
LIN {X 0,Y 196.75,Z 1127.547,A -85,B 0,C 180,E1 9483.987,E2 9483.987} C_VEL
LIN {X 0,Y 186.025,Z 1135.807,A -85,B 0,C 180,E1 9476.839,E2 9476.839} C_VEL
LIN {X 0,Y 179.283,Z 1141.291,A -85,B 0,C 180,E1 9470.57,E2 9470.57} C_VEL
LIN {X 0,Y 174.162,Z 1145.905,A -85,B 0,C 180,E1 9463.614,E2 9463.614} C_VEL
LIN {X 0,Y 170.555,Z 1149.946,A -85,B 0,C 180,E1 9455.045,E2 9455.045} C_VEL
LIN {X 0,Y 169.275,Z 1152.113,A -85,B 0,C 180,E1 9447.63,E2 9447.63} C_VEL
LIN {X 0,Y 169.047,Z 1153.221,A -85,B 0,C 180,E1 9441.036,E2 9441.036} C_VEL
LIN {X 0,Y 169.379,Z 1153.572,A -85,B 0,C 180,E1 9434.595,E2 9434.595} C_VEL
LIN {X 0,Y 170.674,Z 1153.104,A -85,B 0,C 180,E1 9427.617,E2 9427.617} C_VEL
LIN {X 0,Y 173.567,Z 1151.667,A -85,B 0,C 180,E1 9420.446,E2 9420.446} C_VEL
LIN {X 0,Y 178.633,Z 1149.108,A -85,B 0,C 180,E1 9413.208,E2 9413.208} C_VEL
LIN {X 0,Y 187.787,Z 1144.49,A -85,B 0,C 180,E1 9404.915,E2 9404.915} C_VEL
LIN {X 0,Y 199.02,Z 1138.476,A -85,B 0,C 180,E1 9397.931,E2 9397.931} C_VEL
LIN {X 0,Y 210.253,Z 1132.279,A -85,B 0,C 180,E1 9392.677,E2 9392.677} C_VEL
LIN {X 0,Y 225.226,Z 1123.604,A -85,B 0,C 180,E1 9387.211,E2 9387.211} C_VEL
LIN {X 0,Y 242.304,Z 1112.751,A -85,B 0,C 180,E1 9382.312,E2 9382.312} C_VEL
LIN {X 0,Y 257.236,Z 1102.544,A -85,B 0,C 180,E1 9378.822,E2 9378.822} C_VEL
LIN {X 0,Y 273.136,Z 1090.835,A -85,B 0,C 180,E1 9375.687,E2 9375.687} C_VEL
LIN {X 0,Y 292.811,Z 1074.839,A -85,B 0,C 180,E1 9372.419,E2 9372.419} C_VEL
LIN {X 0,Y 307.886,Z 1061.337,A -85,B 0,C 180,E1 9370.266,E2 9370.266} C_VEL
LIN {X 0,Y 322.884,Z 1046.727,A -85,B 0,C 180,E1 9368.369,E2 9368.369} C_VEL
LIN {X 0,Y 340.415,Z 1027.958,A -85,B 0,C 180,E1 9366.409,E2 9366.409} C_VEL
LIN {X 0,Y 356.212,Z 1008.852,A -85,B 0,C 180,E1 9364.826,E2 9364.826} C_VEL
LIN {X 0,Y 369.196,Z 991.524,A -85,B 0,C 180,E1 9363.647,E2 9363.647} C_VEL
LIN {X 0,Y 383.301,Z 970.646,A -85,B 0,C 180,E1 9362.466,E2 9362.466} C_VEL
LIN {X 0,Y 396.516,Z 948.08,A -85,B 0,C 180,E1 9361.425,E2 9361.425} C_VEL
LIN {X 0,Y 406.654,Z 928.513,A -85,B 0,C 180,E1 9360.682,E2 9360.682} C_VEL
LIN {X 0,Y 415.941,Z 908.186,A -85,B 0,C 180,E1 9360.034,E2 9360.034} C_VEL
LIN {X 0,Y 425.967,Z 882.476,A -85,B 0,C 180,E1 9359.354,E2 9359.354} C_VEL
LIN {X 0,Y 433.431,Z 859.025,A -85,B 0,C 180,E1 9358.856,E2 9358.856} C_VEL
LIN {X 0,Y 438.931,Z 838.055,A -85,B 0,C 180,E1 9358.504,E2 9358.504} C_VEL
LIN {X 0,Y 444.015,Z 813.534,A -85,B 0,C 180,E1 9358.161,E2 9358.161} C_VEL
LIN {X 0,Y 449.136,Z 776.665,A -85,B 0,C 180,E1 9357.719,E2 9357.719} C_VEL
LIN {X 0,Y 451.505,Z 757.499,A -85,B 0,C 180,E1 9357.493,E2 9357.493} C_VEL
LIN {X 0,Y 454.748,Z 757.8,A -85,B 0,C 180,E1 9357.202,E2 9357.202} C_VEL
LIN {X 0,Y 454.748,Z 868.607,A -85,B 0,C 180,E1 9357.202,E2 9357.202} C_VEL
LIN {X 0,Y 442.935,Z 868.607,A -85,B 0,C 180,E1 9357.761,E2 9357.761} C_VEL
LIN {X 0,Y 441.063,Z 866.607,A -85,B 0,C 180,E1 9357.852,E2 9357.852} C_VEL
LIN {X 0,Y 441.063,Z 841.283,A -85,B 0,C 180,E1 9357.852,E2 9357.852} C_VEL
LIN {X 0,Y 438.325,Z 840.641,A -85,B 0,C 180,E1 9357.491,E2 9357.491} C_VEL
LIN {X 0,Y 431.872,Z 864.615,A -85,B 0,C 180,E1 9357.169,E2 9357.169} C_VEL
LIN {X 0,Y 422.629,Z 891.887,A -85,B 0,C 180,E1 9356.727,E2 9356.727} C_VEL
LIN {X 0,Y 414.306,Z 912.494,A -85,B 0,C 180,E1 9356.298,E2 9356.298} C_VEL
LIN {X 0,Y 405.037,Z 932.584,A -85,B 0,C 180,E1 9355.787,E2 9355.787} C_VEL
LIN {X 0,Y 393.388,Z 954.876,A -85,B 0,C 180,E1 9355.09,E2 9355.09} C_VEL
LIN {X 0,Y 378.925,Z 978.859,A -85,B 0,C 180,E1 9354.143,E2 9354.143} C_VEL
LIN {X 0,Y 366.491,Z 997.265,A -85,B 0,C 180,E1 9353.247,E2 9353.247} C_VEL
LIN {X 0,Y 353.21,Z 1015.157,A -85,B 0,C 180,E1 9352.19,E2 9352.19} C_VEL
LIN {X 0,Y 336.844,Z 1035.232,A -85,B 0,C 180,E1 9350.738,E2 9350.738} C_VEL
LIN {X 0,Y 318.884,Z 1054.827,A -85,B 0,C 180,E1 9348.935,E2 9348.935} C_VEL
LIN {X 0,Y 303.531,Z 1070.192,A -85,B 0,C 180,E1 9347.175,E2 9347.175} C_VEL
LIN {X 0,Y 286.782,Z 1085.697,A -85,B 0,C 180,E1 9344.962,E2 9344.962} C_VEL
LIN {X 0,Y 265.518,Z 1103.681,A -85,B 0,C 180,E1 9341.614,E2 9341.614} C_VEL
LIN {X 0,Y 249.273,Z 1116.325,A -85,B 0,C 180,E1 9338.525,E2 9338.525} C_VEL
LIN {X 0,Y 233.503,Z 1127.892,A -85,B 0,C 180,E1 9334.917,E2 9334.917} C_VEL
LIN {X 0,Y 215.348,Z 1140.548,A -85,B 0,C 180,E1 9329.723,E2 9329.723} C_VEL
LIN {X 0,Y 199.463,Z 1150.946,A -85,B 0,C 180,E1 9323.809,E2 9323.809} C_VEL
LIN {X 0,Y 187.92,Z 1158.454,A -85,B 0,C 180,E1 9318.15,E2 9318.15} C_VEL
LIN {X 0,Y 177.428,Z 1165.401,A -85,B 0,C 180,E1 9311.249,E2 9311.249} C_VEL
LIN {X 0,Y 168.074,Z 1172.111,A -85,B 0,C 180,E1 9301.969,E2 9301.969} C_VEL
LIN {X 0,Y 163.161,Z 1176.255,A -85,B 0,C 180,E1 9293.474,E2 9293.474} C_VEL
LIN {X 0,Y 161.162,Z 1178.68,A -85,B 0,C 180,E1 9286.212,E2 9286.212} C_VEL
LIN {X 0,Y 160.657,Z 1180.066,A -85,B 0,C 180,E1 9279.312,E2 9279.312} C_VEL
LIN {X 0,Y 160.835,Z 1180.525,A -85,B 0,C 180,E1 9273.208,E2 9273.208} C_VEL
LIN {X 0,Y 160.894,Z 1180.262,A -85,B 0,C 180,E1 9267.863,E2 9267.863} C_VEL
LIN {X 0,Y 160.743,Z 1179.064,A -85,B 0,C 180,E1 9261.775,E2 9261.775} C_VEL
LIN {X 0,Y 161.255,Z 1176.412,A -85,B 0,C 180,E1 9253.798,E2 9253.798} C_VEL
LIN {X 0,Y 164.008,Z 1171.642,A -85,B 0,C 180,E1 9244.739,E2 9244.739} C_VEL
LIN {X 0,Y 168.558,Z 1166.364,A -85,B 0,C 180,E1 9237.33,E2 9237.33} C_VEL
LIN {X 0,Y 175.269,Z 1159.854,A -85,B 0,C 180,E1 9230.288,E2 9230.288} C_VEL
LIN {X 0,Y 185.048,Z 1151.307,A -85,B 0,C 180,E1 9223.161,E2 9223.161} C_VEL
LIN {X 0,Y 198.526,Z 1139.857,A -85,B 0,C 180,E1 9216.106,E2 9216.106} C_VEL
LIN {X 0,Y 210.571,Z 1129.592,A -85,B 0,C 180,E1 9211.274,E2 9211.274} C_VEL
LIN {X 0,Y 223.461,Z 1118.341,A -85,B 0,C 180,E1 9207.076,E2 9207.076} C_VEL
LIN {X 0,Y 239.64,Z 1103.658,A -85,B 0,C 180,E1 9202.768,E2 9202.768} C_VEL
LIN {X 0,Y 256.308,Z 1087.274,A -85,B 0,C 180,E1 9199.129,E2 9199.129} C_VEL
LIN {X 0,Y 270.181,Z 1072.759,A -85,B 0,C 180,E1 9196.557,E2 9196.557} C_VEL
LIN {X 0,Y 285.112,Z 1056.033,A -85,B 0,C 180,E1 9194.151,E2 9194.151} C_VEL
LIN {X 0,Y 302.293,Z 1034.885,A -85,B 0,C 180,E1 9191.752,E2 9191.752} C_VEL
LIN {X 0,Y 315.385,Z 1017.173,A -85,B 0,C 180,E1 9190.144,E2 9190.144} C_VEL
LIN {X 0,Y 327.366,Z 999.513,A -85,B 0,C 180,E1 9188.81,E2 9188.81} C_VEL
LIN {X 0,Y 341.219,Z 977.05,A -85,B 0,C 180,E1 9187.408,E2 9187.408} C_VEL
LIN {X 0,Y 353.564,Z 954.103,A -85,B 0,C 180,E1 9186.271,E2 9186.271} C_VEL
LIN {X 0,Y 363.097,Z 934.254,A -85,B 0,C 180,E1 9185.464,E2 9185.464} C_VEL
LIN {X 0,Y 371.706,Z 914.067,A -85,B 0,C 180,E1 9184.783,E2 9184.783} C_VEL
LIN {X 0,Y 381.239,Z 888.235,A -85,B 0,C 180,E1 9184.08,E2 9184.08} C_VEL
LIN {X 0,Y 388.728,Z 863.282,A -85,B 0,C 180,E1 9183.561,E2 9183.561} C_VEL
LIN {X 0,Y 394.138,Z 841.316,A -85,B 0,C 180,E1 9183.188,E2 9183.188} C_VEL
LIN {X 0,Y 399.191,Z 814.783,A -85,B 0,C 180,E1 9182.773,E2 9182.773} C_VEL
LIN {X 0,Y 404.393,Z 771.444,A -85,B 0,C 180,E1 9182.18,E2 9182.18} C_VEL
LIN {X 0,Y 420.313,Z 628.03,A -85,B 0,C 180,E1 9180.273,E2 9180.273} C_VEL
LIN {X 0,Y 419.126,Z 624.818,A -85,B 0,C 180,E1 9178.29,E2 9178.29} C_VEL
LIN {X 0,Y 418.366,Z 622.491,A -85,B 0,C 180,E1 9176.437,E2 9176.437} C_VEL
LIN {X 0,Y 417.773,Z 620.792,A -85,B 0,C 180,E1 9172.851,E2 9172.851} C_VEL
LIN {X 0,Y 418.42,Z 622.488,A -85,B 0,C 180,E1 9169.118,E2 9169.118} C_VEL
LIN {X 0,Y 419.505,Z 625.773,A -85,B 0,C 180,E1 9166.7,E2 9166.7} C_VEL
LIN {X 0,Y 399.478,Z 801.411,A -85,B 0,C 180,E1 9164.456,E2 9164.456} C_VEL
LIN {X 0,Y 394.982,Z 828.137,A -85,B 0,C 180,E1 9164.057,E2 9164.057} C_VEL
LIN {X 0,Y 389.04,Z 853.209,A -85,B 0,C 180,E1 9163.579,E2 9163.579} C_VEL
LIN {X 0,Y 382.803,Z 874.677,A -85,B 0,C 180,E1 9163.062,E2 9163.062} C_VEL
LIN {X 0,Y 375.021,Z 897.283,A -85,B 0,C 180,E1 9162.391,E2 9162.391} C_VEL
LIN {X 0,Y 364.825,Z 922.041,A -85,B 0,C 180,E1 9161.489,E2 9161.489} C_VEL
LIN {X 0,Y 355.133,Z 942.377,A -85,B 0,C 180,E1 9160.591,E2 9160.591} C_VEL
LIN {X 0,Y 344.659,Z 961.934,A -85,B 0,C 180,E1 9159.557,E2 9159.557} C_VEL
LIN {X 0,Y 330.553,Z 985.238,A -85,B 0,C 180,E1 9158.053,E2 9158.053} C_VEL
LIN {X 0,Y 317.683,Z 1004.028,A -85,B 0,C 180,E1 9156.556,E2 9156.556} C_VEL
LIN {X 0,Y 305.553,Z 1020.182,A -85,B 0,C 180,E1 9155.015,E2 9155.015} C_VEL
LIN {X 0,Y 291.609,Z 1037.206,A -85,B 0,C 180,E1 9153.059,E2 9153.059} C_VEL
LIN {X 0,Y 274.854,Z 1055.671,A -85,B 0,C 180,E1 9150.392,E2 9150.392} C_VEL
LIN {X 0,Y 260.971,Z 1069.666,A -85,B 0,C 180,E1 9147.856,E2 9147.856} C_VEL
LIN {X 0,Y 246.859,Z 1082.897,A -85,B 0,C 180,E1 9144.889,E2 9144.889} C_VEL
LIN {X 0,Y 230.06,Z 1097.525,A -85,B 0,C 180,E1 9140.678,E2 9140.678} C_VEL
LIN {X 0,Y 215.742,Z 1109.046,A -85,B 0,C 180,E1 9136.301,E2 9136.301} C_VEL
LIN {X 0,Y 203.828,Z 1118.221,A -85,B 0,C 180,E1 9131.846,E2 9131.846} C_VEL
LIN {X 0,Y 190.681,Z 1128.123,A -85,B 0,C 180,E1 9125.594,E2 9125.594} C_VEL
LIN {X 0,Y 179.335,Z 1136.398,A -85,B 0,C 180,E1 9118.288,E2 9118.288} C_VEL
LIN {X 0,Y 172.143,Z 1141.892,A -85,B 0,C 180,E1 9111.822,E2 9111.822} C_VEL
LIN {X 0,Y 166.633,Z 1146.516,A -85,B 0,C 180,E1 9104.597,E2 9104.597} C_VEL
LIN {X 0,Y 162.722,Z 1150.576,A -85,B 0,C 180,E1 9095.642,E2 9095.642} C_VEL
LIN {X 0,Y 161.289,Z 1152.82,A -85,B 0,C 180,E1 9087.513,E2 9087.513} C_VEL
LIN {X 0,Y 161.073,Z 1153.889,A -85,B 0,C 180,E1 9080.762,E2 9080.762} C_VEL
LIN {X 0,Y 161.446,Z 1154.241,A -85,B 0,C 180,E1 9074.187,E2 9074.187} C_VEL
LIN {X 0,Y 162.885,Z 1153.792,A -85,B 0,C 180,E1 9066.867,E2 9066.867} C_VEL
LIN {X 0,Y 166.149,Z 1152.337,A -85,B 0,C 180,E1 9059.235,E2 9059.235} C_VEL
LIN {X 0,Y 171.576,Z 1149.831,A -85,B 0,C 180,E1 9051.85,E2 9051.85} C_VEL
LIN {X 0,Y 180.954,Z 1145.476,A -85,B 0,C 180,E1 9043.627,E2 9043.627} C_VEL
LIN {X 0,Y 193.299,Z 1139.25,A -85,B 0,C 180,E1 9036.203,E2 9036.203} C_VEL
LIN {X 0,Y 205.735,Z 1132.734,A -85,B 0,C 180,E1 9030.66,E2 9030.66} C_VEL
LIN {X 0,Y 222.048,Z 1123.68,A -85,B 0,C 180,E1 9025.042,E2 9025.042} C_VEL
LIN {X 0,Y 239.026,Z 1113.207,A -85,B 0,C 180,E1 9020.445,E2 9020.445} C_VEL
LIN {X 0,Y 254.18,Z 1103.156,A -85,B 0,C 180,E1 9017.083,E2 9017.083} C_VEL
LIN {X 0,Y 271.558,Z 1090.681,A -85,B 0,C 180,E1 9013.847,E2 9013.847} C_VEL
LIN {X 0,Y 290.208,Z 1075.81,A -85,B 0,C 180,E1 9010.913,E2 9010.913} C_VEL
LIN {X 0,Y 305.574,Z 1062.35,A -85,B 0,C 180,E1 9008.824,E2 9008.824} C_VEL
LIN {X 0,Y 320.37,Z 1048.245,A -85,B 0,C 180,E1 9007.04,E2 9007.04} C_VEL
LIN {X 0,Y 337.354,Z 1030.518,A -85,B 0,C 180,E1 9005.224,E2 9005.224} C_VEL
LIN {X 0,Y 354.154,Z 1010.681,A -85,B 0,C 180,E1 9003.614,E2 9003.614} C_VEL
LIN {X 0,Y 367.291,Z 993.48,A -85,B 0,C 180,E1 9002.476,E2 9002.476} C_VEL
LIN {X 0,Y 379.612,Z 975.653,A -85,B 0,C 180,E1 9001.482,E2 9001.482} C_VEL
LIN {X 0,Y 393.954,Z 952.273,A -85,B 0,C 180,E1 9000.407,E2 9000.407} C_VEL
LIN {X 0,Y 405.453,Z 930.571,A -85,B 0,C 180,E1 8999.6,E2 8999.6} C_VEL
LIN {X 0,Y 414.505,Z 911.196,A -85,B 0,C 180,E1 8998.998,E2 8998.998} C_VEL
LIN {X 0,Y 423.654,Z 888.694,A -85,B 0,C 180,E1 8998.405,E2 8998.405} C_VEL
LIN {X 0,Y 432.621,Z 861.79,A -85,B 0,C 180,E1 8997.84,E2 8997.84} C_VEL
LIN {X 0,Y 438.325,Z 840.641,A -85,B 0,C 180,E1 8997.491,E2 8997.491} C_VEL
LIN {X 0,Y 441.917,Z 841.152,A -85,B 0,C 180,E1 8997.283,E2 8997.283} C_VEL
LIN {X 0,Y 441.917,Z 919.544,A -85,B 0,C 180,E1 8997.283,E2 8997.283} C_VEL
LIN {X 0,Y 423.741,Z 919.544,A -85,B 0,C 180,E1 8997.832,E2 8997.832} C_VEL
LIN {X 0,Y 421.793,Z 917.544,A -85,B 0,C 180,E1 8997.894,E2 8997.894} C_VEL
LIN {X 0,Y 421.793,Z 902.971,A -85,B 0,C 180,E1 8997.894,E2 8997.894} C_VEL
LIN {X 0,Y 418.474,Z 902.158,A -85,B 0,C 180,E1 8997.634,E2 8997.634} C_VEL
LIN {X 0,Y 407.123,Z 927.59,A -85,B 0,C 180,E1 8997.059,E2 8997.059} C_VEL
LIN {X 0,Y 396.687,Z 947.912,A -85,B 0,C 180,E1 8996.492,E2 8996.492} C_VEL
LIN {X 0,Y 384.98,Z 968.194,A -85,B 0,C 180,E1 8995.799,E2 8995.799} C_VEL
LIN {X 0,Y 368.995,Z 992.594,A -85,B 0,C 180,E1 8994.752,E2 8994.752} C_VEL
LIN {X 0,Y 355.071,Z 1011.411,A -85,B 0,C 180,E1 8993.734,E2 8993.734} C_VEL
LIN {X 0,Y 341.272,Z 1028.412,A -85,B 0,C 180,E1 8992.629,E2 8992.629} C_VEL
LIN {X 0,Y 325.761,Z 1045.898,A -85,B 0,C 180,E1 8991.233,E2 8991.233} C_VEL
LIN {X 0,Y 305.436,Z 1066.528,A -85,B 0,C 180,E1 8989.132,E2 8989.132} C_VEL
LIN {X 0,Y 289.177,Z 1081.502,A -85,B 0,C 180,E1 8987.173,E2 8987.173} C_VEL
LIN {X 0,Y 273.027,Z 1095.271,A -85,B 0,C 180,E1 8984.929,E2 8984.929} C_VEL
LIN {X 0,Y 253.732,Z 1110.551,A -85,B 0,C 180,E1 8981.748,E2 8981.748} C_VEL
LIN {X 0,Y 234.306,Z 1124.53,A -85,B 0,C 180,E1 8977.821,E2 8977.821} C_VEL
LIN {X 0,Y 218.365,Z 1135.316,A -85,B 0,C 180,E1 8973.826,E2 8973.826} C_VEL
LIN {X 0,Y 202.949,Z 1145.25,A -85,B 0,C 180,E1 8969.008,E2 8969.008} C_VEL
LIN {X 0,Y 185.113,Z 1156.274,A -85,B 0,C 180,E1 8961.554,E2 8961.554} C_VEL
LIN {X 0,Y 173.397,Z 1163.439,A -85,B 0,C 180,E1 8954.708,E2 8954.708} C_VEL
LIN {X 0,Y 164.525,Z 1169.084,A -85,B 0,C 180,E1 8947.425,E2 8947.425} C_VEL
LIN {X 0,Y 157.706,Z 1173.936,A -85,B 0,C 180,E1 8938.806,E2 8938.806} C_VEL
LIN {X 0,Y 153.617,Z 1177.676,A -85,B 0,C 180,E1 8928.598,E2 8928.598} C_VEL
LIN {X 0,Y 152.684,Z 1179.37,A -85,B 0,C 180,E1 8920.184,E2 8920.184} C_VEL
LIN {X 0,Y 152.84,Z 1179.864,A -85,B 0,C 180,E1 8913.751,E2 8913.751} C_VEL
LIN {X 0,Y 152.926,Z 1179.614,A -85,B 0,C 180,E1 8908.127,E2 8908.127} C_VEL
LIN {X 0,Y 152.765,Z 1178.438,A -85,B 0,C 180,E1 8901.721,E2 8901.721} C_VEL
LIN {X 0,Y 153.333,Z 1175.803,A -85,B 0,C 180,E1 8893.327,E2 8893.327} C_VEL
LIN {X 0,Y 156.334,Z 1171.065,A -85,B 0,C 180,E1 8883.814,E2 8883.814} C_VEL
LIN {X 0,Y 161.251,Z 1165.797,A -85,B 0,C 180,E1 8876.079,E2 8876.079} C_VEL
LIN {X 0,Y 168.119,Z 1159.573,A -85,B 0,C 180,E1 8869.055,E2 8869.055} C_VEL
LIN {X 0,Y 177.327,Z 1151.94,A -85,B 0,C 180,E1 8862.385,E2 8862.385} C_VEL
LIN {X 0,Y 191.139,Z 1140.884,A -85,B 0,C 180,E1 8855.13,E2 8855.13} C_VEL
LIN {X 0,Y 204.892,Z 1129.654,A -85,B 0,C 180,E1 8849.701,E2 8849.701} C_VEL
LIN {X 0,Y 218.217,Z 1118.483,A -85,B 0,C 180,E1 8845.493,E2 8845.493} C_VEL
LIN {X 0,Y 233.307,Z 1105.25,A -85,B 0,C 180,E1 8841.57,E2 8841.57} C_VEL
LIN {X 0,Y 251.805,Z 1087.818,A -85,B 0,C 180,E1 8837.64,E2 8837.64} C_VEL
LIN {X 0,Y 266.13,Z 1073.256,A -85,B 0,C 180,E1 8835.082,E2 8835.082} C_VEL
LIN {X 0,Y 280.046,Z 1058.1,A -85,B 0,C 180,E1 8832.916,E2 8832.916} C_VEL
LIN {X 0,Y 296.435,Z 1038.828,A -85,B 0,C 180,E1 8830.691,E2 8830.691} C_VEL
LIN {X 0,Y 311.847,Z 1018.54,A -85,B 0,C 180,E1 8828.853,E2 8828.853} C_VEL
LIN {X 0,Y 323.78,Z 1001.385,A -85,B 0,C 180,E1 8827.577,E2 8827.577} C_VEL
LIN {X 0,Y 335.758,Z 982.506,A -85,B 0,C 180,E1 8826.401,E2 8826.401} C_VEL
LIN {X 0,Y 348.856,Z 959.608,A -85,B 0,C 180,E1 8825.237,E2 8825.237} C_VEL
LIN {X 0,Y 360.652,Z 935.688,A -85,B 0,C 180,E1 8824.274,E2 8824.274} C_VEL
LIN {X 0,Y 369.674,Z 914.948,A -85,B 0,C 180,E1 8823.595,E2 8823.595} C_VEL
LIN {X 0,Y 378.894,Z 890.592,A -85,B 0,C 180,E1 8822.948,E2 8822.948} C_VEL
LIN {X 0,Y 387.068,Z 864.104,A -85,B 0,C 180,E1 8822.41,E2 8822.41} C_VEL
LIN {X 0,Y 392.624,Z 841.964,A -85,B 0,C 180,E1 8822.047,E2 8822.047} C_VEL
LIN {X 0,Y 397.271,Z 818.276,A -85,B 0,C 180,E1 8821.686,E2 8821.686} C_VEL
LIN {X 0,Y 401.952,Z 782.651,A -85,B 0,C 180,E1 8821.202,E2 8821.202} C_VEL
LIN {X 0,Y 418.647,Z 634.334,A -85,B 0,C 180,E1 8819.247,E2 8819.247} C_VEL
LIN {X 0,Y 417.329,Z 630.363,A -85,B 0,C 180,E1 8816.291,E2 8816.291} C_VEL
LIN {X 0,Y 416.795,Z 628.735,A -85,B 0,C 180,E1 8812.834,E2 8812.834} C_VEL
LIN {X 0,Y 417.446,Z 630.47,A -85,B 0,C 180,E1 8809.092,E2 8809.092} C_VEL
LIN {X 0,Y 417.958,Z 632.508,A -85,B 0,C 180,E1 8807.709,E2 8807.709} C_VEL
LIN {X 0,Y 398.335,Z 801.938,A -85,B 0,C 180,E1 8805.59,E2 8805.59} C_VEL
LIN {X 0,Y 393.727,Z 828.875,A -85,B 0,C 180,E1 8805.2,E2 8805.2} C_VEL
LIN {X 0,Y 387.784,Z 853.671,A -85,B 0,C 180,E1 8804.744,E2 8804.744} C_VEL
LIN {X 0,Y 381.525,Z 874.998,A -85,B 0,C 180,E1 8804.248,E2 8804.248} C_VEL
LIN {X 0,Y 373.649,Z 897.633,A -85,B 0,C 180,E1 8803.601,E2 8803.601} C_VEL
LIN {X 0,Y 363.025,Z 923.067,A -85,B 0,C 180,E1 8802.706,E2 8802.706} C_VEL
LIN {X 0,Y 353.51,Z 942.765,A -85,B 0,C 180,E1 8801.866,E2 8801.866} C_VEL
LIN {X 0,Y 342.894,Z 962.335,A -85,B 0,C 180,E1 8800.867,E2 8800.867} C_VEL
LIN {X 0,Y 328.892,Z 985.202,A -85,B 0,C 180,E1 8799.446,E2 8799.446} C_VEL
LIN {X 0,Y 315.504,Z 1004.463,A -85,B 0,C 180,E1 8797.965,E2 8797.965} C_VEL
LIN {X 0,Y 303.16,Z 1020.631,A -85,B 0,C 180,E1 8796.473,E2 8796.473} C_VEL
LIN {X 0,Y 288.95,Z 1037.669,A -85,B 0,C 180,E1 8794.574,E2 8794.574} C_VEL
LIN {X 0,Y 271.839,Z 1056.154,A -85,B 0,C 180,E1 8791.975,E2 8791.975} C_VEL
LIN {X 0,Y 257.622,Z 1070.162,A -85,B 0,C 180,E1 8789.497,E2 8789.497} C_VEL
LIN {X 0,Y 243.153,Z 1083.393,A -85,B 0,C 180,E1 8786.589,E2 8786.589} C_VEL
LIN {X 0,Y 225.811,Z 1098.069,A -85,B 0,C 180,E1 8782.428,E2 8782.428} C_VEL
LIN {X 0,Y 210.846,Z 1109.698,A -85,B 0,C 180,E1 8778.036,E2 8778.036} C_VEL
LIN {X 0,Y 198.561,Z 1118.787,A -85,B 0,C 180,E1 8773.619,E2 8773.619} C_VEL
LIN {X 0,Y 185.279,Z 1128.317,A -85,B 0,C 180,E1 8767.575,E2 8767.575} C_VEL
LIN {X 0,Y 173.18,Z 1136.707,A -85,B 0,C 180,E1 8760.152,E2 8760.152} C_VEL
LIN {X 0,Y 165.092,Z 1142.493,A -85,B 0,C 180,E1 8753.182,E2 8753.182} C_VEL
LIN {X 0,Y 159.158,Z 1147.125,A -85,B 0,C 180,E1 8745.672,E2 8745.672} C_VEL
LIN {X 0,Y 154.909,Z 1151.205,A -85,B 0,C 180,E1 8736.299,E2 8736.299} C_VEL
LIN {X 0,Y 153.334,Z 1153.458,A -85,B 0,C 180,E1 8727.757,E2 8727.757} C_VEL
LIN {X 0,Y 153.099,Z 1154.516,A -85,B 0,C 180,E1 8720.982,E2 8720.982} C_VEL
LIN {X 0,Y 153.518,Z 1154.91,A -85,B 0,C 180,E1 8713.736,E2 8713.736} C_VEL
LIN {X 0,Y 155.122,Z 1154.48,A -85,B 0,C 180,E1 8706.041,E2 8706.041} C_VEL
LIN {X 0,Y 158.721,Z 1153.043,A -85,B 0,C 180,E1 8698.051,E2 8698.051} C_VEL
LIN {X 0,Y 164.62,Z 1150.556,A -85,B 0,C 180,E1 8690.376,E2 8690.376} C_VEL
LIN {X 0,Y 174.679,Z 1146.224,A -85,B 0,C 180,E1 8681.916,E2 8681.916} C_VEL
LIN {X 0,Y 187.792,Z 1140.011,A -85,B 0,C 180,E1 8674.36,E2 8674.36} C_VEL
LIN {X 0,Y 200.46,Z 1133.714,A -85,B 0,C 180,E1 8668.936,E2 8668.936} C_VEL
LIN {X 0,Y 216.179,Z 1125.367,A -85,B 0,C 180,E1 8663.683,E2 8663.683} C_VEL
LIN {X 0,Y 234.566,Z 1114.569,A -85,B 0,C 180,E1 8658.863,E2 8658.863} C_VEL
LIN {X 0,Y 250.957,Z 1104.04,A -85,B 0,C 180,E1 8655.383,E2 8655.383} C_VEL
LIN {X 0,Y 267.269,Z 1092.656,A -85,B 0,C 180,E1 8652.471,E2 8652.471} C_VEL
LIN {X 0,Y 287.81,Z 1076.791,A -85,B 0,C 180,E1 8649.382,E2 8649.382} C_VEL
LIN {X 0,Y 303.459,Z 1063.374,A -85,B 0,C 180,E1 8647.362,E2 8647.362} C_VEL
LIN {X 0,Y 318.497,Z 1049.309,A -85,B 0,C 180,E1 8645.64,E2 8645.64} C_VEL
LIN {X 0,Y 334.761,Z 1032.642,A -85,B 0,C 180,E1 8643.983,E2 8643.983} C_VEL
LIN {X 0,Y 352.746,Z 1011.899,A -85,B 0,C 180,E1 8642.346,E2 8642.346} C_VEL
LIN {X 0,Y 366.063,Z 994.727,A -85,B 0,C 180,E1 8641.252,E2 8641.252} C_VEL
LIN {X 0,Y 377.953,Z 977.811,A -85,B 0,C 180,E1 8640.34,E2 8640.34} C_VEL
LIN {X 0,Y 391.468,Z 956.421,A -85,B 0,C 180,E1 8639.376,E2 8639.376} C_VEL
LIN {X 0,Y 404.075,Z 933.312,A -85,B 0,C 180,E1 8638.535,E2 8638.535} C_VEL
LIN {X 0,Y 413.744,Z 913.007,A -85,B 0,C 180,E1 8637.923,E2 8637.923} C_VEL
LIN {X 0,Y 418.474,Z 902.158,A -85,B 0,C 180,E1 8637.634,E2 8637.634} C_VEL
LIN {X 0,Y 421.946,Z 902.953,A -85,B 0,C 180,E1 8637.412,E2 8637.412} C_VEL
LIN {X 0,Y 421.946,Z 959.046,A -85,B 0,C 180,E1 8637.412,E2 8637.412} C_VEL
LIN {X 0,Y 403.583,Z 959.046,A -85,B 0,C 180,E1 8637.881,E2 8637.881} C_VEL
LIN {X 0,Y 401.618,Z 957.046,A -85,B 0,C 180,E1 8637.933,E2 8637.933} C_VEL
LIN {X 0,Y 401.618,Z 945.798,A -85,B 0,C 180,E1 8637.933,E2 8637.933} C_VEL
LIN {X 0,Y 398.109,Z 944.79,A -85,B 0,C 180,E1 8637.753,E2 8637.753} C_VEL
LIN {X 0,Y 386.926,Z 964.288,A -85,B 0,C 180,E1 8637.144,E2 8637.144} C_VEL
LIN {X 0,Y 374.68,Z 983.439,A -85,B 0,C 180,E1 8636.417,E2 8636.417} C_VEL
LIN {X 0,Y 358.685,Z 1005.809,A -85,B 0,C 180,E1 8635.363,E2 8635.363} C_VEL
LIN {X 0,Y 342.23,Z 1026.085,A -85,B 0,C 180,E1 8634.156,E2 8634.156} C_VEL
LIN {X 0,Y 327.051,Z 1043.107,A -85,B 0,C 180,E1 8632.891,E2 8632.891} C_VEL
LIN {X 0,Y 309.568,Z 1061.034,A -85,B 0,C 180,E1 8631.24,E2 8631.24} C_VEL
LIN {X 0,Y 289.546,Z 1079.421,A -85,B 0,C 180,E1 8629.051,E2 8629.051} C_VEL
LIN {X 0,Y 273.029,Z 1093.302,A -85,B 0,C 180,E1 8626.936,E2 8626.936} C_VEL
LIN {X 0,Y 255.797,Z 1106.706,A -85,B 0,C 180,E1 8624.353,E2 8624.353} C_VEL
LIN {X 0,Y 234.495,Z 1121.97,A -85,B 0,C 180,E1 8620.444,E2 8620.444} C_VEL
LIN {X 0,Y 216.508,Z 1133.772,A -85,B 0,C 180,E1 8616.31,E2 8616.31} C_VEL
LIN {X 0,Y 201.525,Z 1143.061,A -85,B 0,C 180,E1 8612.024,E2 8612.024} C_VEL
LIN {X 0,Y 186.034,Z 1152.251,A -85,B 0,C 180,E1 8606.385,E2 8606.385} C_VEL
LIN {X 0,Y 169.477,Z 1161.757,A -85,B 0,C 180,E1 8598.019,E2 8598.019} C_VEL
LIN {X 0,Y 159.08,Z 1167.805,A -85,B 0,C 180,E1 8590.345,E2 8590.345} C_VEL
LIN {X 0,Y 151.734,Z 1172.404,A -85,B 0,C 180,E1 8582.26,E2 8582.26} C_VEL
LIN {X 0,Y 146.926,Z 1175.986,A -85,B 0,C 180,E1 8573.247,E2 8573.247} C_VEL
LIN {X 0,Y 144.843,Z 1178.391,A -85,B 0,C 180,E1 8563.574,E2 8563.574} C_VEL
LIN {X 0,Y 144.795,Z 1179.22,A -85,B 0,C 180,E1 8555.548,E2 8555.548} C_VEL
LIN {X 0,Y 144.974,Z 1179.026,A -85,B 0,C 180,E1 8549.605,E2 8549.605} C_VEL
LIN {X 0,Y 144.84,Z 1178.194,A -85,B 0,C 180,E1 8543.659,E2 8543.659} C_VEL
LIN {X 0,Y 144.885,Z 1176.616,A -85,B 0,C 180,E1 8537.242,E2 8537.242} C_VEL
LIN {X 0,Y 146.118,Z 1173.812,A -85,B 0,C 180,E1 8529.575,E2 8529.575} C_VEL
LIN {X 0,Y 149.313,Z 1169.787,A -85,B 0,C 180,E1 8521.612,E2 8521.612} C_VEL
LIN {X 0,Y 154.726,Z 1164.6,A -85,B 0,C 180,E1 8513.881,E2 8513.881} C_VEL
LIN {X 0,Y 162.593,Z 1158.078,A -85,B 0,C 180,E1 8506.47,E2 8506.47} C_VEL
LIN {X 0,Y 174.915,Z 1148.619,A -85,B 0,C 180,E1 8498.453,E2 8498.453} C_VEL
LIN {X 0,Y 188.675,Z 1138.029,A -85,B 0,C 180,E1 8492.003,E2 8492.003} C_VEL
LIN {X 0,Y 201.474,Z 1128.04,A -85,B 0,C 180,E1 8487.337,E2 8487.337} C_VEL
LIN {X 0,Y 216.171,Z 1116.131,A -85,B 0,C 180,E1 8483.011,E2 8483.011} C_VEL
LIN {X 0,Y 235.159,Z 1099.742,A -85,B 0,C 180,E1 8478.53,E2 8478.53} C_VEL
LIN {X 0,Y 250.191,Z 1085.725,A -85,B 0,C 180,E1 8475.608,E2 8475.608} C_VEL
LIN {X 0,Y 264.907,Z 1071.029,A -85,B 0,C 180,E1 8473.149,E2 8473.149} C_VEL
LIN {X 0,Y 281.871,Z 1052.767,A -85,B 0,C 180,E1 8470.712,E2 8470.712} C_VEL
LIN {X 0,Y 298.356,Z 1032.982,A -85,B 0,C 180,E1 8468.657,E2 8468.657} C_VEL
LIN {X 0,Y 311.696,Z 1015.468,A -85,B 0,C 180,E1 8467.187,E2 8467.187} C_VEL
LIN {X 0,Y 324.674,Z 996.814,A -85,B 0,C 180,E1 8465.902,E2 8465.902} C_VEL
LIN {X 0,Y 340.009,Z 972.062,A -85,B 0,C 180,E1 8464.522,E2 8464.522} C_VEL
LIN {X 0,Y 351.149,Z 951.656,A -85,B 0,C 180,E1 8463.616,E2 8463.616} C_VEL
LIN {X 0,Y 360.415,Z 932.695,A -85,B 0,C 180,E1 8462.917,E2 8462.917} C_VEL
LIN {X 0,Y 369.734,Z 911.176,A -85,B 0,C 180,E1 8462.262,E2 8462.262} C_VEL
LIN {X 0,Y 379.843,Z 883.545,A -85,B 0,C 180,E1 8461.601,E2 8461.601} C_VEL
LIN {X 0,Y 386.589,Z 861.186,A -85,B 0,C 180,E1 8461.188,E2 8461.188} C_VEL
LIN {X 0,Y 392.157,Z 838.691,A -85,B 0,C 180,E1 8460.839,E2 8460.839} C_VEL
LIN {X 0,Y 397.453,Z 810.033,A -85,B 0,C 180,E1 8460.425,E2 8460.425} C_VEL
LIN {X 0,Y 404.172,Z 753.835,A -85,B 0,C 180,E1 8459.696,E2 8459.696} C_VEL
LIN {X 0,Y 417.11,Z 640.865,A -85,B 0,C 180,E1 8458.249,E2 8458.249} C_VEL
LIN {X 0,Y 416.295,Z 638.236,A -85,B 0,C 180,E1 8456.144,E2 8456.144} C_VEL
LIN {X 0,Y 415.816,Z 636.679,A -85,B 0,C 180,E1 8452.817,E2 8452.817} C_VEL
LIN {X 0,Y 416.42,Z 638.368,A -85,B 0,C 180,E1 8449.205,E2 8449.205} C_VEL
LIN {X 0,Y 416.542,Z 639.24,A -85,B 0,C 180,E1 8448.726,E2 8448.726} C_VEL
LIN {X 0,Y 397.362,Z 802.354,A -85,B 0,C 180,E1 8446.733,E2 8446.733} C_VEL
LIN {X 0,Y 392.686,Z 829.337,A -85,B 0,C 180,E1 8446.354,E2 8446.354} C_VEL
LIN {X 0,Y 386.68,Z 854.12,A -85,B 0,C 180,E1 8445.915,E2 8445.915} C_VEL
LIN {X 0,Y 380.309,Z 875.58,A -85,B 0,C 180,E1 8445.435,E2 8445.435} C_VEL
LIN {X 0,Y 371.99,Z 899.169,A -85,B 0,C 180,E1 8444.783,E2 8444.783} C_VEL
LIN {X 0,Y 361.486,Z 923.869,A -85,B 0,C 180,E1 8443.942,E2 8443.942} C_VEL
LIN {X 0,Y 352.064,Z 943.15,A -85,B 0,C 180,E1 8443.151,E2 8443.151} C_VEL
LIN {X 0,Y 341.756,Z 961.955,A -85,B 0,C 180,E1 8442.231,E2 8442.231} C_VEL
LIN {X 0,Y 328.442,Z 983.688,A -85,B 0,C 180,E1 8440.95,E2 8440.95} C_VEL
LIN {X 0,Y 313.953,Z 1004.316,A -85,B 0,C 180,E1 8439.441,E2 8439.441} C_VEL
LIN {X 0,Y 301.395,Z 1020.55,A -85,B 0,C 180,E1 8438.005,E2 8438.005} C_VEL
LIN {X 0,Y 287.339,Z 1037.162,A -85,B 0,C 180,E1 8436.228,E2 8436.228} C_VEL
LIN {X 0,Y 269.037,Z 1056.637,A -85,B 0,C 180,E1 8433.593,E2 8433.593} C_VEL
LIN {X 0,Y 254.491,Z 1070.657,A -85,B 0,C 180,E1 8431.179,E2 8431.179} C_VEL
LIN {X 0,Y 239.644,Z 1083.901,A -85,B 0,C 180,E1 8428.336,E2 8428.336} C_VEL
LIN {X 0,Y 221.778,Z 1098.602,A -85,B 0,C 180,E1 8424.243,E2 8424.243} C_VEL
LIN {X 0,Y 206.421,Z 1110.154,A -85,B 0,C 180,E1 8419.935,E2 8419.935} C_VEL
LIN {X 0,Y 193.494,Z 1119.352,A -85,B 0,C 180,E1 8415.487,E2 8415.487} C_VEL
LIN {X 0,Y 179.567,Z 1128.892,A -85,B 0,C 180,E1 8409.403,E2 8409.403} C_VEL
LIN {X 0,Y 166.775,Z 1137.3,A -85,B 0,C 180,E1 8401.842,E2 8401.842} C_VEL
LIN {X 0,Y 158.14,Z 1143.095,A -85,B 0,C 180,E1 8394.663,E2 8394.663} C_VEL
LIN {X 0,Y 151.74,Z 1147.737,A -85,B 0,C 180,E1 8386.853,E2 8386.853} C_VEL
LIN {X 0,Y 147.118,Z 1151.834,A -85,B 0,C 180,E1 8377.026,E2 8377.026} C_VEL
LIN {X 0,Y 145.381,Z 1154.096,A -85,B 0,C 180,E1 8368.029,E2 8368.029} C_VEL
LIN {X 0,Y 145.124,Z 1155.167,A -85,B 0,C 180,E1 8360.882,E2 8360.882} C_VEL
LIN {X 0,Y 145.594,Z 1155.579,A -85,B 0,C 180,E1 8353.236,E2 8353.236} C_VEL
LIN {X 0,Y 147.392,Z 1155.168,A -85,B 0,C 180,E1 8345.128,E2 8345.128} C_VEL
LIN {X 0,Y 151.365,Z 1153.75,A -85,B 0,C 180,E1 8336.752,E2 8336.752} C_VEL
LIN {X 0,Y 157.777,Z 1151.281,A -85,B 0,C 180,E1 8328.771,E2 8328.771} C_VEL
LIN {X 0,Y 168.567,Z 1146.968,A -85,B 0,C 180,E1 8320.078,E2 8320.078} C_VEL
LIN {X 0,Y 182.435,Z 1140.804,A -85,B 0,C 180,E1 8312.433,E2 8312.433} C_VEL
LIN {X 0,Y 195.497,Z 1134.635,A -85,B 0,C 180,E1 8307.078,E2 8307.078} C_VEL
LIN {X 0,Y 210.591,Z 1126.963,A -85,B 0,C 180,E1 8302.205,E2 8302.205} C_VEL
LIN {X 0,Y 231.112,Z 1115.43,A -85,B 0,C 180,E1 8297.038,E2 8297.038} C_VEL
LIN {X 0,Y 247.098,Z 1105.487,A -85,B 0,C 180,E1 8293.8,E2 8293.8} C_VEL
LIN {X 0,Y 262.874,Z 1094.823,A -85,B 0,C 180,E1 8291.092,E2 8291.092} C_VEL
LIN {X 0,Y 281.003,Z 1081.447,A -85,B 0,C 180,E1 8288.439,E2 8288.439} C_VEL
LIN {X 0,Y 300.599,Z 1065.238,A -85,B 0,C 180,E1 8285.99,E2 8285.99} C_VEL
LIN {X 0,Y 316.126,Z 1051.036,A -85,B 0,C 180,E1 8284.296,E2 8284.296} C_VEL
LIN {X 0,Y 331.353,Z 1035.779,A -85,B 0,C 180,E1 8282.813,E2 8282.813} C_VEL
LIN {X 0,Y 348.579,Z 1016.733,A -85,B 0,C 180,E1 8281.315,E2 8281.315} C_VEL
LIN {X 0,Y 364.449,Z 996.727,A -85,B 0,C 180,E1 8280.063,E2 8280.063} C_VEL
LIN {X 0,Y 376.988,Z 979.2,A -85,B 0,C 180,E1 8279.152,E2 8279.152} C_VEL
LIN {X 0,Y 389.11,Z 960.362,A -85,B 0,C 180,E1 8278.329,E2 8278.329} C_VEL
LIN {X 0,Y 398.109,Z 944.79,A -85,B 0,C 180,E1 8277.753,E2 8277.753} C_VEL
LIN {X 0,Y 401.313,Z 945.875,A -85,B 0,C 180,E1 8277.493,E2 8277.493} C_VEL
LIN {X 0,Y 401.313,Z 991.713,A -85,B 0,C 180,E1 8277.493,E2 8277.493} C_VEL
LIN {X 0,Y 382.645,Z 991.713,A -85,B 0,C 180,E1 8278.09,E2 8278.09} C_VEL
LIN {X 0,Y 380.694,Z 989.713,A -85,B 0,C 180,E1 8278.156,E2 8278.156} C_VEL
LIN {X 0,Y 380.694,Z 979.605,A -85,B 0,C 180,E1 8278.156,E2 8278.156} C_VEL
LIN {X 0,Y 377.722,Z 978.358,A -85,B 0,C 180,E1 8277.859,E2 8277.859} C_VEL
LIN {X 0,Y 364.915,Z 996.666,A -85,B 0,C 180,E1 8277.102,E2 8277.102} C_VEL
LIN {X 0,Y 350.732,Z 1015.029,A -85,B 0,C 180,E1 8276.174,E2 8276.174} C_VEL
LIN {X 0,Y 332.226,Z 1036.495,A -85,B 0,C 180,E1 8274.82,E2 8274.82} C_VEL
LIN {X 0,Y 315.806,Z 1053.532,A -85,B 0,C 180,E1 8273.455,E2 8273.455} C_VEL
LIN {X 0,Y 299.915,Z 1068.664,A -85,B 0,C 180,E1 8271.948,E2 8271.948} C_VEL
LIN {X 0,Y 283.157,Z 1083.346,A -85,B 0,C 180,E1 8270.124,E2 8270.124} C_VEL
LIN {X 0,Y 261.342,Z 1100.715,A -85,B 0,C 180,E1 8267.316,E2 8267.316} C_VEL
LIN {X 0,Y 242.872,Z 1114.02,A -85,B 0,C 180,E1 8264.437,E2 8264.437} C_VEL
LIN {X 0,Y 225.959,Z 1125.331,A -85,B 0,C 180,E1 8261.252,E2 8261.252} C_VEL
LIN {X 0,Y 206.746,Z 1137.345,A -85,B 0,C 180,E1 8256.762,E2 8256.762} C_VEL
LIN {X 0,Y 187.63,Z 1148.32,A -85,B 0,C 180,E1 8250.92,E2 8250.92} C_VEL
LIN {X 0,Y 173.203,Z 1156.22,A -85,B 0,C 180,E1 8245.058,E2 8245.058} C_VEL
LIN {X 0,Y 160.75,Z 1162.902,A -85,B 0,C 180,E1 8238.275,E2 8238.275} C_VEL
LIN {X 0,Y 148.757,Z 1169.554,A -85,B 0,C 180,E1 8228.689,E2 8228.689} C_VEL
LIN {X 0,Y 141.095,Z 1174.112,A -85,B 0,C 180,E1 8218.346,E2 8218.346} C_VEL
LIN {X 0,Y 137.742,Z 1176.709,A -85,B 0,C 180,E1 8209.319,E2 8209.319} C_VEL
LIN {X 0,Y 136.745,Z 1178.055,A -85,B 0,C 180,E1 8201.386,E2 8201.386} C_VEL
LIN {X 0,Y 136.878,Z 1178.517,A -85,B 0,C 180,E1 8194.189,E2 8194.189} C_VEL
LIN {X 0,Y 136.984,Z 1178.295,A -85,B 0,C 180,E1 8188.327,E2 8188.327} C_VEL
LIN {X 0,Y 136.809,Z 1177.185,A -85,B 0,C 180,E1 8181.595,E2 8181.595} C_VEL
LIN {X 0,Y 137.443,Z 1174.712,A -85,B 0,C 180,E1 8172.647,E2 8172.647} C_VEL
LIN {X 0,Y 141.121,Z 1169.901,A -85,B 0,C 180,E1 8161.66,E2 8161.66} C_VEL
LIN {X 0,Y 146.894,Z 1164.662,A -85,B 0,C 180,E1 8153.203,E2 8153.203} C_VEL
LIN {X 0,Y 154.72,Z 1158.529,A -85,B 0,C 180,E1 8145.739,E2 8145.739} C_VEL
LIN {X 0,Y 165.193,Z 1150.855,A -85,B 0,C 180,E1 8138.667,E2 8138.667} C_VEL
LIN {X 0,Y 180.282,Z 1140.033,A -85,B 0,C 180,E1 8131.341,E2 8131.341} C_VEL
LIN {X 0,Y 195.722,Z 1128.467,A -85,B 0,C 180,E1 8125.737,E2 8125.737} C_VEL
LIN {X 0,Y 209.817,Z 1117.504,A -85,B 0,C 180,E1 8121.682,E2 8121.682} C_VEL
LIN {X 0,Y 225.064,Z 1104.989,A -85,B 0,C 180,E1 8118.066,E2 8118.066} C_VEL
LIN {X 0,Y 244.535,Z 1087.765,A -85,B 0,C 180,E1 8114.293,E2 8114.293} C_VEL
LIN {X 0,Y 260.397,Z 1072.415,A -85,B 0,C 180,E1 8111.726,E2 8111.726} C_VEL
LIN {X 0,Y 274.886,Z 1057.297,A -85,B 0,C 180,E1 8109.695,E2 8109.695} C_VEL
LIN {X 0,Y 291.56,Z 1038.417,A -85,B 0,C 180,E1 8107.66,E2 8107.66} C_VEL
LIN {X 0,Y 308.084,Z 1017.41,A -85,B 0,C 180,E1 8105.894,E2 8105.894} C_VEL
LIN {X 0,Y 321.018,Z 999.29,A -85,B 0,C 180,E1 8104.668,E2 8104.668} C_VEL
LIN {X 0,Y 333.6,Z 979.86,A -85,B 0,C 180,E1 8103.572,E2 8103.572} C_VEL
LIN {X 0,Y 348.261,Z 954.218,A -85,B 0,C 180,E1 8102.422,E2 8102.422} C_VEL
LIN {X 0,Y 358.431,Z 933.864,A -85,B 0,C 180,E1 8101.693,E2 8101.693} C_VEL
LIN {X 0,Y 367.471,Z 913.425,A -85,B 0,C 180,E1 8101.091,E2 8101.091} C_VEL
LIN {X 0,Y 377.209,Z 888.035,A -85,B 0,C 180,E1 8100.491,E2 8100.491} C_VEL
LIN {X 0,Y 385.163,Z 862.333,A -85,B 0,C 180,E1 8100.027,E2 8100.027} C_VEL
LIN {X 0,Y 390.731,Z 840.364,A -85,B 0,C 180,E1 8099.7,E2 8099.7} C_VEL
LIN {X 0,Y 395.876,Z 814.266,A -85,B 0,C 180,E1 8099.331,E2 8099.331} C_VEL
LIN {X 0,Y 401.044,Z 773.616,A -85,B 0,C 180,E1 8098.812,E2 8098.812} C_VEL
LIN {X 0,Y 415.664,Z 647.591,A -85,B 0,C 180,E1 8097.242,E2 8097.242} C_VEL
LIN {X 0,Y 415.222,Z 646.022,A -85,B 0,C 180,E1 8095.857,E2 8095.857} C_VEL
LIN {X 0,Y 414.838,Z 644.622,A -85,B 0,C 180,E1 8092.8,E2 8092.8} C_VEL
LIN {X 0,Y 415.243,Z 646.095,A -85,B 0,C 180,E1 8089.748,E2 8089.748} C_VEL
LIN {X 0,Y 396.549,Z 802.769,A -85,B 0,C 180,E1 8087.88,E2 8087.88} C_VEL
LIN {X 0,Y 391.805,Z 829.798,A -85,B 0,C 180,E1 8087.514,E2 8087.514} C_VEL
LIN {X 0,Y 385.753,Z 854.523,A -85,B 0,C 180,E1 8087.094,E2 8087.094} C_VEL
LIN {X 0,Y 379.229,Z 876.249,A -85,B 0,C 180,E1 8086.627,E2 8086.627} C_VEL
LIN {X 0,Y 370.49,Z 900.698,A -85,B 0,C 180,E1 8085.976,E2 8085.976} C_VEL
LIN {X 0,Y 359.931,Z 925.037,A -85,B 0,C 180,E1 8085.175,E2 8085.175} C_VEL
LIN {X 0,Y 350.34,Z 944.365,A -85,B 0,C 180,E1 8084.41,E2 8084.41} C_VEL
LIN {X 0,Y 339.004,Z 964.673,A -85,B 0,C 180,E1 8083.446,E2 8083.446} C_VEL
LIN {X 0,Y 323.725,Z 988.615,A -85,B 0,C 180,E1 8082.042,E2 8082.042} C_VEL
LIN {X 0,Y 311.285,Z 1005.922,A -85,B 0,C 180,E1 8080.792,E2 8080.792} C_VEL
LIN {X 0,Y 298.704,Z 1021.866,A -85,B 0,C 180,E1 8079.422,E2 8079.422} C_VEL
LIN {X 0,Y 283.404,Z 1039.564,A -85,B 0,C 180,E1 8077.569,E2 8077.569} C_VEL
LIN {X 0,Y 265.618,Z 1057.927,A -85,B 0,C 180,E1 8075.119,E2 8075.119} C_VEL
LIN {X 0,Y 250.772,Z 1071.887,A -85,B 0,C 180,E1 8072.763,E2 8072.763} C_VEL
LIN {X 0,Y 235.045,Z 1085.533,A -85,B 0,C 180,E1 8069.869,E2 8069.869} C_VEL
LIN {X 0,Y 215.747,Z 1100.763,A -85,B 0,C 180,E1 8065.58,E2 8065.58} C_VEL
LIN {X 0,Y 201.029,Z 1111.438,A -85,B 0,C 180,E1 8061.557,E2 8061.557} C_VEL
LIN {X 0,Y 186.722,Z 1121.209,A -85,B 0,C 180,E1 8056.74,E2 8056.74} C_VEL
LIN {X 0,Y 170.152,Z 1131.88,A -85,B 0,C 180,E1 8049.393,E2 8049.393} C_VEL
LIN {X 0,Y 159.141,Z 1138.745,A -85,B 0,C 180,E1 8042.705,E2 8042.705} C_VEL
LIN {X 0,Y 150.218,Z 1144.411,A -85,B 0,C 180,E1 8035.213,E2 8035.213} C_VEL
LIN {X 0,Y 142.712,Z 1149.667,A -85,B 0,C 180,E1 8025.44,E2 8025.44} C_VEL
LIN {X 0,Y 138.727,Z 1152.993,A -85,B 0,C 180,E1 8015.791,E2 8015.791} C_VEL
LIN {X 0,Y 137.393,Z 1154.801,A -85,B 0,C 180,E1 8007.914,E2 8007.914} C_VEL
LIN {X 0,Y 137.152,Z 1155.847,A -85,B 0,C 180,E1 8000.347,E2 8000.347} C_VEL
LIN {X 0,Y 137.741,Z 1156.238,A -85,B 0,C 180,E1 7992.249,E2 7992.249} C_VEL
LIN {X 0,Y 139.851,Z 1155.807,A -85,B 0,C 180,E1 7983.687,E2 7983.687} C_VEL
LIN {X 0,Y 144.364,Z 1154.365,A -85,B 0,C 180,E1 7974.91,E2 7974.91} C_VEL
LIN {X 0,Y 151.867,Z 1151.728,A -85,B 0,C 180,E1 7966.267,E2 7966.267} C_VEL
LIN {X 0,Y 164.789,Z 1146.818,A -85,B 0,C 180,E1 7956.782,E2 7956.782} C_VEL
LIN {X 0,Y 178.614,Z 1141.016,A -85,B 0,C 180,E1 7949.811,E2 7949.811} C_VEL
LIN {X 0,Y 193.112,Z 1134.46,A -85,B 0,C 180,E1 7944.32,E2 7944.32} C_VEL
LIN {X 0,Y 212.256,Z 1124.956,A -85,B 0,C 180,E1 7938.766,E2 7938.766} C_VEL
LIN {X 0,Y 230.442,Z 1114.787,A -85,B 0,C 180,E1 7934.631,E2 7934.631} C_VEL
LIN {X 0,Y 246.968,Z 1104.696,A -85,B 0,C 180,E1 7931.551,E2 7931.551} C_VEL
LIN {X 0,Y 266.867,Z 1091.375,A -85,B 0,C 180,E1 7928.46,E2 7928.46} C_VEL
LIN {X 0,Y 286.477,Z 1076.475,A -85,B 0,C 180,E1 7925.899,E2 7925.899} C_VEL
LIN {X 0,Y 302.722,Z 1062.899,A -85,B 0,C 180,E1 7924.073,E2 7924.073} C_VEL
LIN {X 0,Y 319.242,Z 1047.743,A -85,B 0,C 180,E1 7922.43,E2 7922.43} C_VEL
LIN {X 0,Y 338.48,Z 1027.965,A -85,B 0,C 180,E1 7920.738,E2 7920.738} C_VEL
LIN {X 0,Y 352.959,Z 1011.3,A -85,B 0,C 180,E1 7919.592,E2 7919.592} C_VEL
LIN {X 0,Y 366.05,Z 994.687,A -85,B 0,C 180,E1 7918.646,E2 7918.646} C_VEL
LIN {X 0,Y 377.722,Z 978.358,A -85,B 0,C 180,E1 7917.859,E2 7917.859} C_VEL
LIN {X 0,Y 373.369,Z 984.926,A -85,B 0,C 180,E1 7917.568,E2 7917.568} C_VEL
LIN {X 0,Y 367.862,Z 992.622,A -85,B 0,C 180,E1 7917.51,E2 7917.51} C_VEL
LIN {X 0,Y 360.412,Z 1002.456,A -85,B 0,C 180,E1 7917.773,E2 7917.773} C_VEL
LIN {X 0,Y 349.904,Z 1015.197,A -85,B 0,C 180,E1 7918.467,E2 7918.467} C_VEL
LIN {X 0,Y 330.954,Z 1035.986,A -85,B 0,C 180,E1 7919.908,E2 7919.908} C_VEL
LIN {X 0,Y 314.966,Z 1051.64,A -85,B 0,C 180,E1 7921.273,E2 7921.273} C_VEL
LIN {X 0,Y 299.307,Z 1065.604,A -85,B 0,C 180,E1 7922.768,E2 7922.768} C_VEL
LIN {X 0,Y 279.561,Z 1081.579,A -85,B 0,C 180,E1 7924.924,E2 7924.924} C_VEL
LIN {X 0,Y 260.132,Z 1095.423,A -85,B 0,C 180,E1 7927.402,E2 7927.402} C_VEL
LIN {X 0,Y 243.252,Z 1106.36,A -85,B 0,C 180,E1 7929.941,E2 7929.941} C_VEL
LIN {X 0,Y 225.807,Z 1116.659,A -85,B 0,C 180,E1 7933.057,E2 7933.057} C_VEL
LIN {X 0,Y 203.63,Z 1128.339,A -85,B 0,C 180,E1 7938.02,E2 7938.02} C_VEL
LIN {X 0,Y 187.461,Z 1135.929,A -85,B 0,C 180,E1 7942.671,E2 7942.671} C_VEL
LIN {X 0,Y 172.453,Z 1142.364,A -85,B 0,C 180,E1 7948.203,E2 7948.203} C_VEL
LIN {X 0,Y 156.361,Z 1148.647,A -85,B 0,C 180,E1 7956.32,E2 7956.32} C_VEL
LIN {X 0,Y 144.511,Z 1152.735,A -85,B 0,C 180,E1 7965.111,E2 7965.111} C_VEL
LIN {X 0,Y 136.914,Z 1155.167,A -85,B 0,C 180,E1 7973.734,E2 7973.734} C_VEL
LIN {X 0,Y 131.876,Z 1156.602,A -85,B 0,C 180,E1 7983.468,E2 7983.468} C_VEL
LIN {X 0,Y 129.566,Z 1156.949,A -85,B 0,C 180,E1 7993.87,E2 7993.87} C_VEL
LIN {X 0,Y 129.195,Z 1156.271,A -85,B 0,C 180,E1 8002.887,E2 8002.887} C_VEL
LIN {X 0,Y 129.966,Z 1154.7,A -85,B 0,C 180,E1 8012.204,E2 8012.204} C_VEL
LIN {X 0,Y 132.738,Z 1152.068,A -85,B 0,C 180,E1 8021.734,E2 8021.734} C_VEL
LIN {X 0,Y 137.692,Z 1148.578,A -85,B 0,C 180,E1 8030.399,E2 8030.399} C_VEL
LIN {X 0,Y 145.396,Z 1143.828,A -85,B 0,C 180,E1 8038.775,E2 8038.775} C_VEL
LIN {X 0,Y 157.526,Z 1136.767,A -85,B 0,C 180,E1 8047.541,E2 8047.541} C_VEL
LIN {X 0,Y 171.772,Z 1128.125,A -85,B 0,C 180,E1 8054.774,E2 8054.774} C_VEL
LIN {X 0,Y 185.378,Z 1119.596,A -85,B 0,C 180,E1 8059.986,E2 8059.986} C_VEL
LIN {X 0,Y 201.644,Z 1108.801,A -85,B 0,C 180,E1 8064.9,E2 8064.9} C_VEL
LIN {X 0,Y 219.829,Z 1095.544,A -85,B 0,C 180,E1 8069.276,E2 8069.276} C_VEL
LIN {X 0,Y 234.944,Z 1083.582,A -85,B 0,C 180,E1 8072.275,E2 8072.275} C_VEL
LIN {X 0,Y 249.749,Z 1070.913,A -85,B 0,C 180,E1 8074.793,E2 8074.793} C_VEL
LIN {X 0,Y 267.527,Z 1054.354,A -85,B 0,C 180,E1 8077.389,E2 8077.389} C_VEL
LIN {X 0,Y 283.979,Z 1037.116,A -85,B 0,C 180,E1 8079.48,E2 8079.48} C_VEL
LIN {X 0,Y 297.639,Z 1021.445,A -85,B 0,C 180,E1 8081.021,E2 8081.021} C_VEL
LIN {X 0,Y 311.035,Z 1004.589,A -85,B 0,C 180,E1 8082.389,E2 8082.389} C_VEL
LIN {X 0,Y 326.334,Z 983.168,A -85,B 0,C 180,E1 8083.81,E2 8083.81} C_VEL
LIN {X 0,Y 339.15,Z 962.695,A -85,B 0,C 180,E1 8084.908,E2 8084.908} C_VEL
LIN {X 0,Y 349.707,Z 943.846,A -85,B 0,C 180,E1 8085.752,E2 8085.752} C_VEL
LIN {X 0,Y 360.332,Z 922.463,A -85,B 0,C 180,E1 8086.55,E2 8086.55} C_VEL
LIN {X 0,Y 371.006,Z 897.284,A -85,B 0,C 180,E1 8087.313,E2 8087.313} C_VEL
LIN {X 0,Y 378.72,Z 875.681,A -85,B 0,C 180,E1 8087.852,E2 8087.852} C_VEL
LIN {X 0,Y 385.325,Z 853.724,A -85,B 0,C 180,E1 8088.301,E2 8088.301} C_VEL
LIN {X 0,Y 391.755,Z 827.018,A -85,B 0,C 180,E1 8088.725,E2 8088.725} C_VEL
LIN {X 0,Y 396.08,Z 801.868,A -85,B 0,C 180,E1 8089.047,E2 8089.047} C_VEL
LIN {X 0,Y 414.023,Z 653.367,A -85,B 0,C 180,E1 8090.788,E2 8090.788} C_VEL
LIN {X 0,Y 413.861,Z 652.598,A -85,B 0,C 180,E1 8093.201,E2 8093.201} C_VEL
LIN {X 0,Y 414.335,Z 654.361,A -85,B 0,C 180,E1 8096.221,E2 8096.221} C_VEL
LIN {X 0,Y 396.293,Z 805.815,A -85,B 0,C 180,E1 8098.068,E2 8098.068} C_VEL
LIN {X 0,Y 391.538,Z 833.055,A -85,B 0,C 180,E1 8098.427,E2 8098.427} C_VEL
LIN {X 0,Y 385.218,Z 858.744,A -85,B 0,C 180,E1 8098.789,E2 8098.789} C_VEL
LIN {X 0,Y 378.738,Z 880.167,A -85,B 0,C 180,E1 8099.134,E2 8099.134} C_VEL
LIN {X 0,Y 369.954,Z 904.67,A -85,B 0,C 180,E1 8099.636,E2 8099.636} C_VEL
LIN {X 0,Y 358.953,Z 930.087,A -85,B 0,C 180,E1 8100.306,E2 8100.306} C_VEL
LIN {X 0,Y 348.999,Z 950.154,A -85,B 0,C 180,E1 8100.966,E2 8100.966} C_VEL
LIN {X 0,Y 337.754,Z 970.355,A -85,B 0,C 180,E1 8101.772,E2 8101.772} C_VEL
LIN {X 0,Y 321.936,Z 995.364,A -85,B 0,C 180,E1 8103.027,E2 8103.027} C_VEL
LIN {X 0,Y 308.776,Z 1013.815,A -85,B 0,C 180,E1 8104.178,E2 8104.178} C_VEL
LIN {X 0,Y 295.314,Z 1031.043,A -85,B 0,C 180,E1 8105.494,E2 8105.494} C_VEL
LIN {X 0,Y 278.731,Z 1050.423,A -85,B 0,C 180,E1 8107.32,E2 8107.32} C_VEL
LIN {X 0,Y 260.626,Z 1069.29,A -85,B 0,C 180,E1 8109.618,E2 8109.618} C_VEL
LIN {X 0,Y 246.127,Z 1083.198,A -85,B 0,C 180,E1 8111.755,E2 8111.755} C_VEL
LIN {X 0,Y 231.136,Z 1096.565,A -85,B 0,C 180,E1 8114.308,E2 8114.308} C_VEL
LIN {X 0,Y 212.516,Z 1112.048,A -85,B 0,C 180,E1 8118.126,E2 8118.126} C_VEL
LIN {X 0,Y 194.888,Z 1125.401,A -85,B 0,C 180,E1 8122.631,E2 8122.631} C_VEL
LIN {X 0,Y 180.866,Z 1135.503,A -85,B 0,C 180,E1 8127.123,E2 8127.123} C_VEL
LIN {X 0,Y 167.344,Z 1144.895,A -85,B 0,C 180,E1 8132.6,E2 8132.6} C_VEL
LIN {X 0,Y 152.781,Z 1154.942,A -85,B 0,C 180,E1 8140.611,E2 8140.611} C_VEL
LIN {X 0,Y 141.609,Z 1162.777,A -85,B 0,C 180,E1 8149.693,E2 8149.693} C_VEL
LIN {X 0,Y 134.848,Z 1168.157,A -85,B 0,C 180,E1 8158.235,E2 8158.235} C_VEL
LIN {X 0,Y 130.768,Z 1172.259,A -85,B 0,C 180,E1 8167.049,E2 8167.049} C_VEL
LIN {X 0,Y 129.086,Z 1175.01,A -85,B 0,C 180,E1 8175.191,E2 8175.191} C_VEL
LIN {X 0,Y 128.849,Z 1176.713,A -85,B 0,C 180,E1 8182.42,E2 8182.42} C_VEL
LIN {X 0,Y 129.024,Z 1177.666,A -85,B 0,C 180,E1 8189.112,E2 8189.112} C_VEL
LIN {X 0,Y 128.858,Z 1177.862,A -85,B 0,C 180,E1 8195.343,E2 8195.343} C_VEL
LIN {X 0,Y 128.902,Z 1177.223,A -85,B 0,C 180,E1 8203.914,E2 8203.914} C_VEL
LIN {X 0,Y 131.314,Z 1175.166,A -85,B 0,C 180,E1 8214.758,E2 8214.758} C_VEL
LIN {X 0,Y 137.862,Z 1171.208,A -85,B 0,C 180,E1 8225.977,E2 8225.977} C_VEL
LIN {X 0,Y 146.623,Z 1166.654,A -85,B 0,C 180,E1 8234.619,E2 8234.619} C_VEL
LIN {X 0,Y 158.066,Z 1160.942,A -85,B 0,C 180,E1 8242.251,E2 8242.251} C_VEL
LIN {X 0,Y 174.468,Z 1152.722,A -85,B 0,C 180,E1 8249.925,E2 8249.925} C_VEL
LIN {X 0,Y 193.361,Z 1142.561,A -85,B 0,C 180,E1 8256.242,E2 8256.242} C_VEL
LIN {X 0,Y 210.267,Z 1132.896,A -85,B 0,C 180,E1 8260.557,E2 8260.557} C_VEL
LIN {X 0,Y 228.514,Z 1121.712,A -85,B 0,C 180,E1 8264.282,E2 8264.282} C_VEL
LIN {X 0,Y 252.093,Z 1105.816,A -85,B 0,C 180,E1 8268.097,E2 8268.097} C_VEL
LIN {X 0,Y 269.727,Z 1092.714,A -85,B 0,C 180,E1 8270.416,E2 8270.416} C_VEL
LIN {X 0,Y 286.541,Z 1079.151,A -85,B 0,C 180,E1 8272.303,E2 8272.303} C_VEL
LIN {X 0,Y 304.599,Z 1063.293,A -85,B 0,C 180,E1 8274.048,E2 8274.048} C_VEL
LIN {X 0,Y 324.854,Z 1043.458,A -85,B 0,C 180,E1 8275.734,E2 8275.734} C_VEL
LIN {X 0,Y 340.459,Z 1026.497,A -85,B 0,C 180,E1 8276.871,E2 8276.871} C_VEL
LIN {X 0,Y 355.206,Z 1008.89,A -85,B 0,C 180,E1 8277.823,E2 8277.823} C_VEL
LIN {X 0,Y 357.176,Z 1006.444,A -85,B 0,C 180,E1 8277.961,E2 8277.961} C_VEL
LIN {X 0,Y 349.904,Z 1015.197,A -85,B 0,C 180,E1 8278.467,E2 8278.467} C_VEL
LIN {X 0,Y 345.637,Z 1020.239,A -85,B 0,C 180,E1 8278.608,E2 8278.608} C_VEL
LIN {X 0,Y 340.489,Z 1026.064,A -85,B 0,C 180,E1 8278.457,E2 8278.457} C_VEL
LIN {X 0,Y 330.044,Z 1037.409,A -85,B 0,C 180,E1 8277.628,E2 8277.628} C_VEL
LIN {X 0,Y 326.224,Z 1041.38,A -85,B 0,C 180,E1 8277.323,E2 8277.323} C_VEL
LIN {X 0,Y 306.762,Z 1060.509,A -85,B 0,C 180,E1 8275.849,E2 8275.849} C_VEL
LIN {X 0,Y 286.498,Z 1078.117,A -85,B 0,C 180,E1 8274.06,E2 8274.06} C_VEL
LIN {X 0,Y 268.457,Z 1092.42,A -85,B 0,C 180,E1 8272.184,E2 8272.184} C_VEL
LIN {X 0,Y 248.004,Z 1107.262,A -85,B 0,C 180,E1 8269.647,E2 8269.647} C_VEL
LIN {X 0,Y 225.482,Z 1121.856,A -85,B 0,C 180,E1 8266.196,E2 8266.196} C_VEL
LIN {X 0,Y 207.337,Z 1132.617,A -85,B 0,C 180,E1 8262.714,E2 8262.714} C_VEL
LIN {X 0,Y 188.51,Z 1142.958,A -85,B 0,C 180,E1 8258.157,E2 8258.157} C_VEL
LIN {X 0,Y 167.522,Z 1153.522,A -85,B 0,C 180,E1 8251.327,E2 8251.327} C_VEL
LIN {X 0,Y 152.412,Z 1160.676,A -85,B 0,C 180,E1 8244.436,E2 8244.436} C_VEL
LIN {X 0,Y 140.236,Z 1166.315,A -85,B 0,C 180,E1 8236.656,E2 8236.656} C_VEL
LIN {X 0,Y 129.138,Z 1171.693,A -85,B 0,C 180,E1 8225.61,E2 8225.61} C_VEL
LIN {X 0,Y 122.8,Z 1175.107,A -85,B 0,C 180,E1 8213.514,E2 8213.514} C_VEL
LIN {X 0,Y 120.915,Z 1176.651,A -85,B 0,C 180,E1 8203.875,E2 8203.875} C_VEL
LIN {X 0,Y 120.891,Z 1177.179,A -85,B 0,C 180,E1 8195.22,E2 8195.22} C_VEL
LIN {X 0,Y 121.05,Z 1176.996,A -85,B 0,C 180,E1 8189.054,E2 8189.054} C_VEL
LIN {X 0,Y 120.871,Z 1176.085,A -85,B 0,C 180,E1 8182.395,E2 8182.395} C_VEL
LIN {X 0,Y 121.209,Z 1174.269,A -85,B 0,C 180,E1 8174.204,E2 8174.204} C_VEL
LIN {X 0,Y 123.273,Z 1171.381,A -85,B 0,C 180,E1 8165.293,E2 8165.293} C_VEL
LIN {X 0,Y 127.803,Z 1167.338,A -85,B 0,C 180,E1 8156.258,E2 8156.258} C_VEL
LIN {X 0,Y 135.443,Z 1161.813,A -85,B 0,C 180,E1 8147.223,E2 8147.223} C_VEL
LIN {X 0,Y 148.525,Z 1153.27,A -85,B 0,C 180,E1 8137.405,E2 8137.405} C_VEL
LIN {X 0,Y 162.893,Z 1143.914,A -85,B 0,C 180,E1 8130.064,E2 8130.064} C_VEL
LIN {X 0,Y 177.122,Z 1134.481,A -85,B 0,C 180,E1 8124.654,E2 8124.654} C_VEL
LIN {X 0,Y 194.234,Z 1122.61,A -85,B 0,C 180,E1 8119.606,E2 8119.606} C_VEL
LIN {X 0,Y 213.41,Z 1108.152,A -85,B 0,C 180,E1 8115.173,E2 8115.173} C_VEL
LIN {X 0,Y 229.161,Z 1095.355,A -85,B 0,C 180,E1 8112.222,E2 8112.222} C_VEL
LIN {X 0,Y 244.521,Z 1081.927,A -85,B 0,C 180,E1 8109.784,E2 8109.784} C_VEL
LIN {X 0,Y 262.143,Z 1065.237,A -85,B 0,C 180,E1 8107.396,E2 8107.396} C_VEL
LIN {X 0,Y 280.64,Z 1045.698,A -85,B 0,C 180,E1 8105.257,E2 8105.257} C_VEL
LIN {X 0,Y 294.62,Z 1029.477,A -85,B 0,C 180,E1 8103.845,E2 8103.845} C_VEL
LIN {X 0,Y 308.273,Z 1012.16,A -85,B 0,C 180,E1 8102.602,E2 8102.602} C_VEL
LIN {X 0,Y 324.04,Z 990.062,A -85,B 0,C 180,E1 8101.327,E2 8101.327} C_VEL
LIN {X 0,Y 337.956,Z 967.731,A -85,B 0,C 180,E1 8100.313,E2 8100.313} C_VEL
LIN {X 0,Y 348.959,Z 947.985,A -85,B 0,C 180,E1 8099.581,E2 8099.581} C_VEL
LIN {X 0,Y 360.377,Z 924.869,A -85,B 0,C 180,E1 8098.887,E2 8098.887} C_VEL
LIN {X 0,Y 370.77,Z 900.016,A -85,B 0,C 180,E1 8098.3,E2 8098.3} C_VEL
LIN {X 0,Y 378.471,Z 878.397,A -85,B 0,C 180,E1 8097.896,E2 8097.896} C_VEL
LIN {X 0,Y 385.167,Z 856.123,A -85,B 0,C 180,E1 8097.566,E2 8097.566} C_VEL
LIN {X 0,Y 391.935,Z 827.387,A -85,B 0,C 180,E1 8097.183,E2 8097.183} C_VEL
LIN {X 0,Y 395.966,Z 803.552,A -85,B 0,C 180,E1 8096.883,E2 8096.883} C_VEL
LIN {X 0,Y 413.082,Z 661.538,A -85,B 0,C 180,E1 8095.175,E2 8095.175} C_VEL
LIN {X 0,Y 412.882,Z 660.531,A -85,B 0,C 180,E1 8092.626,E2 8092.626} C_VEL
LIN {X 0,Y 412.899,Z 660.963,A -85,B 0,C 180,E1 8091.796,E2 8091.796} C_VEL
LIN {X 0,Y 395.401,Z 803.601,A -85,B 0,C 180,E1 8090.187,E2 8090.187} C_VEL
LIN {X 0,Y 390.541,Z 830.666,A -85,B 0,C 180,E1 8089.848,E2 8089.848} C_VEL
LIN {X 0,Y 384.362,Z 855.428,A -85,B 0,C 180,E1 8089.465,E2 8089.465} C_VEL
LIN {X 0,Y 377.831,Z 876.786,A -85,B 0,C 180,E1 8089.045,E2 8089.045} C_VEL
LIN {X 0,Y 369.381,Z 900.049,A -85,B 0,C 180,E1 8088.486,E2 8088.486} C_VEL
LIN {X 0,Y 358.603,Z 924.729,A -85,B 0,C 180,E1 8087.759,E2 8087.759} C_VEL
LIN {X 0,Y 348.336,Z 945.061,A -85,B 0,C 180,E1 8087.031,E2 8087.031} C_VEL
LIN {X 0,Y 337.201,Z 964.622,A -85,B 0,C 180,E1 8086.189,E2 8086.189} C_VEL
LIN {X 0,Y 321.999,Z 988.114,A -85,B 0,C 180,E1 8084.95,E2 8084.95} C_VEL
LIN {X 0,Y 308.297,Z 1006.752,A -85,B 0,C 180,E1 8083.734,E2 8083.734} C_VEL
LIN {X 0,Y 294.727,Z 1023.468,A -85,B 0,C 180,E1 8082.418,E2 8082.418} C_VEL
